(* IEC 61131-3 sources: OpenPLC-Simulator/openplc/OpenPLC/src (part 2) *)

(* ---- SIM_FB_RunTasks.st ---- *)
(* ============================================================
   SIM_FB_RunTasks.st — Simulate transporter task execution

   For each active transporter [1..3], checks whether a new task
   has been assigned (task_id <> running_task_id) and executes
   the full transport cycle:

     Phase 0  idle        — waiting for new task
     Phase 1  to_lift     — X-drive towards lift station
     Phase 2  lifting     — Z-lift sequence (stages 1-5)
     Phase 3  to_sink     — X-drive towards sink station
     Phase 4  sinking     — Z-sink sequence (stages 6-8)

   Also maintains current_station (nearest station) every cycle.

   Called once per PLC scan from PLC_PRG.
   ============================================================ *)

FUNCTION_BLOCK SIM_FB_RunTasks
VAR_INPUT
  i_run : BOOL;       (* enable — typically init_done *)
END_VAR
VAR_EXTERNAL CONSTANT
    TRANSPORTERS : INT;
END_VAR

VAR_EXTERNAL
  g_transporter  : ARRAY[1..TRANSPORTERS] OF STC_TRANSPORTER_T;
  g_stations     : ARRAY[101..125] OF STATION_T;
  g_cfg          : ARRAY[1..TRANSPORTERS] OF TRANSPORTER_CFG_T;
  g_move         : ARRAY[1..TRANSPORTERS] OF MOVE_TIMES_T;
END_VAR
VAR
  i            : INT;
  idx          : INT;
  (* Physics FB instances — one per transporter (MATIEC needs separate instances) *)
  fb_x1        : SIM_FB_XMotion;
  fb_x2        : SIM_FB_XMotion;
  fb_x3        : SIM_FB_XMotion;
  fb_z1        : SIM_FB_ZMotion;
  fb_z2        : SIM_FB_ZMotion;
  fb_z3        : SIM_FB_ZMotion;
  (* Station lookup *)
  lookup       : STC_FB_FindStation;
  (* Temp vars for VAR_IN_OUT passing *)
  tmp_x        : REAL;
  tmp_vx       : REAL;
  tmp_z        : REAL;
  tmp_zs       : INT;
  tmp_zt       : REAL;
  arrived_x    : BOOL;
  at_station   : BOOL;    (* TRUE only when actually at station, not just at drive limit *)
  arrived_z    : BOOL;
  station_type : INT;
  device_delay : REAL;
  drop_time    : REAL;
  (* Nearest-station calculation *)
  nearest_num  : INT;
  min_dist     : REAL;
  dx           : REAL;
  (* Time measurement instances *)
  tm1          : STC_FB_MeasureMoveTimes;
  tm2          : STC_FB_MeasureMoveTimes;
  tm3          : STC_FB_MeasureMoveTimes;
END_VAR

IF NOT i_run THEN
  RETURN;
END_IF;

FOR i := 1 TO TRANSPORTERS DO
  IF g_transporter[i].active THEN

  (* ── Phase 0 → 1: Accept new task ───────────────────────── *)
  IF (g_transporter[i].phase = 0)
     AND (g_transporter[i].task_id <> g_transporter[i].running_task_id) THEN
    g_transporter[i].running_task_id := g_transporter[i].task_id;
    lookup(station_number := g_transporter[i].lift_station);
    g_transporter[i].final_target_x := lookup.x_mm;
    g_transporter[i].phase := 1;
    g_transporter[i].z_stage := 0;
    g_transporter[i].z_timer_s := 0.0;

  (* ── Phase 1: Drive X towards lift station ──────────────── *)
  ELSIF g_transporter[i].phase = 1 THEN
    tmp_x  := g_transporter[i].x_mm;
    tmp_vx := g_transporter[i].vel_x;
    IF i = 1 THEN
      fb_x1(
        delta_t  := 0.02,
        x_target := g_transporter[i].final_target_x,
        x_min    := g_transporter[i].x_min_limit,
        x_max    := g_transporter[i].x_max_limit,
        v_max    := g_cfg[i].phys2d.x_max_mm_s,
        t_acc    := g_cfg[i].phys2d.x_accel_s,
        t_dec    := g_cfg[i].phys2d.x_decel_s,
        x_pos    := tmp_x,
        v_x      := tmp_vx
      );
      arrived_x := fb_x1.arrived;
    ELSIF i = 2 THEN
      fb_x2(
        delta_t  := 0.02,
        x_target := g_transporter[i].final_target_x,
        x_min    := g_transporter[i].x_min_limit,
        x_max    := g_transporter[i].x_max_limit,
        v_max    := g_cfg[i].phys2d.x_max_mm_s,
        t_acc    := g_cfg[i].phys2d.x_accel_s,
        t_dec    := g_cfg[i].phys2d.x_decel_s,
        x_pos    := tmp_x,
        v_x      := tmp_vx
      );
      arrived_x := fb_x2.arrived;
    ELSIF i = 3 THEN
      fb_x3(
        delta_t  := 0.02,
        x_target := g_transporter[i].final_target_x,
        x_min    := g_transporter[i].x_min_limit,
        x_max    := g_transporter[i].x_max_limit,
        v_max    := g_cfg[i].phys2d.x_max_mm_s,
        t_acc    := g_cfg[i].phys2d.x_accel_s,
        t_dec    := g_cfg[i].phys2d.x_decel_s,
        x_pos    := tmp_x,
        v_x      := tmp_vx
      );
      arrived_x := fb_x3.arrived;
    END_IF;
    g_transporter[i].x_mm  := tmp_x;
    g_transporter[i].vel_x := tmp_vx;

    (* Only transition when actually at station, not just at drive limit *)
    at_station := arrived_x
                  AND (ABS(g_transporter[i].x_mm - g_transporter[i].final_target_x) <= 6.0);
    IF at_station THEN
      g_transporter[i].current_station := g_transporter[i].lift_station;
      lookup(station_number := g_transporter[i].lift_station);
      device_delay := lookup.device_delay_s;
      drop_time    := lookup.dropping_time_s;
      g_transporter[i].z_timer_s := device_delay + drop_time;
      g_transporter[i].z_stage := 1;
      g_transporter[i].phase := 2;
    END_IF;
    (* If arrived_x but not at_station → at drive limit, wait for clearance *)

  (* ── Phase 2: Lift Z at lift station ────────────────────── *)
  ELSIF g_transporter[i].phase = 2 THEN
    lookup(station_number := g_transporter[i].lift_station);
    station_type := lookup.stype;
    tmp_z  := g_transporter[i].z_mm;
    tmp_zs := g_transporter[i].z_stage;
    tmp_zt := g_transporter[i].z_timer_s;
    IF i = 1 THEN
      fb_z1(
        delta_t       := 0.02,
        station_type  := station_type,
        z_total_mm    := g_cfg[i].phys2d.z_total_mm,
        z_slow_dry_mm := g_cfg[i].phys2d.z_slow_dry_mm,
        z_slow_wet_mm := g_cfg[i].phys2d.z_slow_wet_mm,
        z_slow_end_mm := g_cfg[i].phys2d.z_slow_end_mm,
        z_slow_mm_s   := g_cfg[i].phys2d.z_slow_mm_s,
        z_fast_mm_s   := g_cfg[i].phys2d.z_fast_mm_s,
        drip_delay_s  := g_cfg[i].phys2d.drip_delay_s,
        z_mm          := tmp_z,
        z_stage       := tmp_zs,
        z_timer_s     := tmp_zt
      );
      arrived_z := fb_z1.done;
    ELSIF i = 2 THEN
      fb_z2(
        delta_t       := 0.02,
        station_type  := station_type,
        z_total_mm    := g_cfg[i].phys2d.z_total_mm,
        z_slow_dry_mm := g_cfg[i].phys2d.z_slow_dry_mm,
        z_slow_wet_mm := g_cfg[i].phys2d.z_slow_wet_mm,
        z_slow_end_mm := g_cfg[i].phys2d.z_slow_end_mm,
        z_slow_mm_s   := g_cfg[i].phys2d.z_slow_mm_s,
        z_fast_mm_s   := g_cfg[i].phys2d.z_fast_mm_s,
        drip_delay_s  := g_cfg[i].phys2d.drip_delay_s,
        z_mm          := tmp_z,
        z_stage       := tmp_zs,
        z_timer_s     := tmp_zt
      );
      arrived_z := fb_z2.done;
    ELSIF i = 3 THEN
      fb_z3(
        delta_t       := 0.02,
        station_type  := station_type,
        z_total_mm    := g_cfg[i].phys2d.z_total_mm,
        z_slow_dry_mm := g_cfg[i].phys2d.z_slow_dry_mm,
        z_slow_wet_mm := g_cfg[i].phys2d.z_slow_wet_mm,
        z_slow_end_mm := g_cfg[i].phys2d.z_slow_end_mm,
        z_slow_mm_s   := g_cfg[i].phys2d.z_slow_mm_s,
        z_fast_mm_s   := g_cfg[i].phys2d.z_fast_mm_s,
        drip_delay_s  := g_cfg[i].phys2d.drip_delay_s,
        z_mm          := tmp_z,
        z_stage       := tmp_zs,
        z_timer_s     := tmp_zt
      );
      arrived_z := fb_z3.done;
    END_IF;
    g_transporter[i].z_mm      := tmp_z;
    g_transporter[i].z_stage   := tmp_zs;
    g_transporter[i].z_timer_s := tmp_zt;
    IF arrived_z THEN
      lookup(station_number := g_transporter[i].sink_station);
      g_transporter[i].final_target_x := lookup.x_mm;
      g_transporter[i].phase := 3;
    END_IF;

  (* ── Phase 3: Drive X towards sink station ─────────────── *)
  ELSIF g_transporter[i].phase = 3 THEN
    tmp_x  := g_transporter[i].x_mm;
    tmp_vx := g_transporter[i].vel_x;
    IF i = 1 THEN
      fb_x1(
        delta_t  := 0.02,
        x_target := g_transporter[i].final_target_x,
        x_min    := g_transporter[i].x_min_limit,
        x_max    := g_transporter[i].x_max_limit,
        v_max    := g_cfg[i].phys2d.x_max_mm_s,
        t_acc    := g_cfg[i].phys2d.x_accel_s,
        t_dec    := g_cfg[i].phys2d.x_decel_s,
        x_pos    := tmp_x,
        v_x      := tmp_vx
      );
      arrived_x := fb_x1.arrived;
    ELSIF i = 2 THEN
      fb_x2(
        delta_t  := 0.02,
        x_target := g_transporter[i].final_target_x,
        x_min    := g_transporter[i].x_min_limit,
        x_max    := g_transporter[i].x_max_limit,
        v_max    := g_cfg[i].phys2d.x_max_mm_s,
        t_acc    := g_cfg[i].phys2d.x_accel_s,
        t_dec    := g_cfg[i].phys2d.x_decel_s,
        x_pos    := tmp_x,
        v_x      := tmp_vx
      );
      arrived_x := fb_x2.arrived;
    ELSIF i = 3 THEN
      fb_x3(
        delta_t  := 0.02,
        x_target := g_transporter[i].final_target_x,
        x_min    := g_transporter[i].x_min_limit,
        x_max    := g_transporter[i].x_max_limit,
        v_max    := g_cfg[i].phys2d.x_max_mm_s,
        t_acc    := g_cfg[i].phys2d.x_accel_s,
        t_dec    := g_cfg[i].phys2d.x_decel_s,
        x_pos    := tmp_x,
        v_x      := tmp_vx
      );
      arrived_x := fb_x3.arrived;
    END_IF;
    g_transporter[i].x_mm  := tmp_x;
    g_transporter[i].vel_x := tmp_vx;

    (* Only transition when actually at station, not just at drive limit *)
    at_station := arrived_x
                  AND (ABS(g_transporter[i].x_mm - g_transporter[i].final_target_x) <= 6.0);
    IF at_station THEN
      g_transporter[i].current_station := g_transporter[i].sink_station;
      lookup(station_number := g_transporter[i].sink_station);
      device_delay := lookup.device_delay_s;
      g_transporter[i].z_timer_s := device_delay + g_cfg[i].phys2d.drip_delay_s;
      g_transporter[i].z_stage := 6;
      g_transporter[i].phase := 4;
    END_IF;
    (* If arrived_x but not at_station → at drive limit, wait for clearance *)

  (* ── Phase 4: Sink Z at sink station ───────────────────── *)
  ELSIF g_transporter[i].phase = 4 THEN
    lookup(station_number := g_transporter[i].sink_station);
    station_type := lookup.stype;
    tmp_z  := g_transporter[i].z_mm;
    tmp_zs := g_transporter[i].z_stage;
    tmp_zt := g_transporter[i].z_timer_s;
    IF i = 1 THEN
      fb_z1(
        delta_t       := 0.02,
        station_type  := station_type,
        z_total_mm    := g_cfg[i].phys2d.z_total_mm,
        z_slow_dry_mm := g_cfg[i].phys2d.z_slow_dry_mm,
        z_slow_wet_mm := g_cfg[i].phys2d.z_slow_wet_mm,
        z_slow_end_mm := g_cfg[i].phys2d.z_slow_end_mm,
        z_slow_mm_s   := g_cfg[i].phys2d.z_slow_mm_s,
        z_fast_mm_s   := g_cfg[i].phys2d.z_fast_mm_s,
        drip_delay_s  := g_cfg[i].phys2d.drip_delay_s,
        z_mm          := tmp_z,
        z_stage       := tmp_zs,
        z_timer_s     := tmp_zt
      );
      arrived_z := fb_z1.done;
    ELSIF i = 2 THEN
      fb_z2(
        delta_t       := 0.02,
        station_type  := station_type,
        z_total_mm    := g_cfg[i].phys2d.z_total_mm,
        z_slow_dry_mm := g_cfg[i].phys2d.z_slow_dry_mm,
        z_slow_wet_mm := g_cfg[i].phys2d.z_slow_wet_mm,
        z_slow_end_mm := g_cfg[i].phys2d.z_slow_end_mm,
        z_slow_mm_s   := g_cfg[i].phys2d.z_slow_mm_s,
        z_fast_mm_s   := g_cfg[i].phys2d.z_fast_mm_s,
        drip_delay_s  := g_cfg[i].phys2d.drip_delay_s,
        z_mm          := tmp_z,
        z_stage       := tmp_zs,
        z_timer_s     := tmp_zt
      );
      arrived_z := fb_z2.done;
    ELSIF i = 3 THEN
      fb_z3(
        delta_t       := 0.02,
        station_type  := station_type,
        z_total_mm    := g_cfg[i].phys2d.z_total_mm,
        z_slow_dry_mm := g_cfg[i].phys2d.z_slow_dry_mm,
        z_slow_wet_mm := g_cfg[i].phys2d.z_slow_wet_mm,
        z_slow_end_mm := g_cfg[i].phys2d.z_slow_end_mm,
        z_slow_mm_s   := g_cfg[i].phys2d.z_slow_mm_s,
        z_fast_mm_s   := g_cfg[i].phys2d.z_fast_mm_s,
        drip_delay_s  := g_cfg[i].phys2d.drip_delay_s,
        z_mm          := tmp_z,
        z_stage       := tmp_zs,
        z_timer_s     := tmp_zt
      );
      arrived_z := fb_z3.done;
    END_IF;
    g_transporter[i].z_mm      := tmp_z;
    g_transporter[i].z_stage   := tmp_zs;
    g_transporter[i].z_timer_s := tmp_zt;
    IF arrived_z THEN
      g_transporter[i].phase := 0;
    END_IF;
  END_IF;  (* ELSIF chain: phases 0→1→2→3→4 *)

  (* ── Phase 0 idle: drive back inside limits if outside ────── *)
  IF g_transporter[i].phase = 0 THEN
    tmp_x  := g_transporter[i].x_mm;
    tmp_vx := g_transporter[i].vel_x;
    (* Use current position as target — XMotion will clamp to nearest limit if outside *)
    IF i = 1 THEN
      fb_x1(
        delta_t  := 0.02,
        x_target := tmp_x,
        x_min    := g_transporter[i].x_min_limit,
        x_max    := g_transporter[i].x_max_limit,
        v_max    := g_cfg[i].phys2d.x_max_mm_s,
        t_acc    := g_cfg[i].phys2d.x_accel_s,
        t_dec    := g_cfg[i].phys2d.x_decel_s,
        x_pos    := tmp_x,
        v_x      := tmp_vx
      );
    ELSIF i = 2 THEN
      fb_x2(
        delta_t  := 0.02,
        x_target := tmp_x,
        x_min    := g_transporter[i].x_min_limit,
        x_max    := g_transporter[i].x_max_limit,
        v_max    := g_cfg[i].phys2d.x_max_mm_s,
        t_acc    := g_cfg[i].phys2d.x_accel_s,
        t_dec    := g_cfg[i].phys2d.x_decel_s,
        x_pos    := tmp_x,
        v_x      := tmp_vx
      );
    ELSIF i = 3 THEN
      fb_x3(
        delta_t  := 0.02,
        x_target := tmp_x,
        x_min    := g_transporter[i].x_min_limit,
        x_max    := g_transporter[i].x_max_limit,
        v_max    := g_cfg[i].phys2d.x_max_mm_s,
        t_acc    := g_cfg[i].phys2d.x_accel_s,
        t_dec    := g_cfg[i].phys2d.x_decel_s,
        x_pos    := tmp_x,
        v_x      := tmp_vx
      );
    END_IF;
    g_transporter[i].x_mm  := tmp_x;
    g_transporter[i].vel_x := tmp_vx;
  END_IF;

  (* ── Nearest station tracking ──────────────────────────── *)
  min_dist := 1.0e9;
  nearest_num := g_transporter[i].current_station;
  FOR idx := 101 TO 125 DO
    IF g_stations[idx].tank_id <> 0 THEN
      dx := g_stations[idx].x_position - g_transporter[i].x_mm;
      IF ABS(dx) < min_dist THEN
        min_dist := ABS(dx);
        nearest_num := idx;
      END_IF;
    END_IF;
  END_FOR;
  g_transporter[i].current_station := nearest_num;

  (* ── Measure move times (one instance per transporter) ──── *)
  IF i = 1 THEN
    tm1(t_id := 1, phase := g_transporter[1].phase, delta_t := 0.02,
        vel_x := g_transporter[1].vel_x, z_stage := g_transporter[1].z_stage,
        lift_stn := g_transporter[1].lift_station,
        sink_stn := g_transporter[1].sink_station,
        from_stn := g_transporter[1].current_station);
  ELSIF i = 2 THEN
    tm2(t_id := 2, phase := g_transporter[2].phase, delta_t := 0.02,
        vel_x := g_transporter[2].vel_x, z_stage := g_transporter[2].z_stage,
        lift_stn := g_transporter[2].lift_station,
        sink_stn := g_transporter[2].sink_station,
        from_stn := g_transporter[2].current_station);
  ELSIF i = 3 THEN
    tm3(t_id := 3, phase := g_transporter[3].phase, delta_t := 0.02,
        vel_x := g_transporter[3].vel_x, z_stage := g_transporter[3].z_stage,
        lift_stn := g_transporter[3].lift_station,
        sink_stn := g_transporter[3].sink_station,
        from_stn := g_transporter[3].current_station);
  END_IF;

  END_IF;  (* active *)
END_FOR;

END_FUNCTION_BLOCK

(* ---- SIM_FB_XMotion.st ---- *)
(* ============================================================
   SIM_FB_XMotion.st — Horizontal motion with accel / decel
   ============================================================ *)

FUNCTION_BLOCK SIM_FB_XMotion
VAR_INPUT
  delta_t  : REAL;
  x_target : REAL;
  x_min    : REAL;
  x_max    : REAL;
  v_max    : REAL;
  t_acc    : REAL;
  t_dec    : REAL;
END_VAR
VAR_IN_OUT
  x_pos : REAL;
  v_x   : REAL;
END_VAR
VAR_OUTPUT
  arrived : BOOL;
END_VAR
VAR
  drive_target : REAL;
  distance     : REAL;
  dir          : REAL;
  a_acc        : REAL;
  a_dec        : REAL;
  brake_dist   : REAL;
  new_vel      : REAL;
  travel       : REAL;
END_VAR
  IF (x_max > x_min) THEN
    IF x_pos < x_min THEN
      drive_target := x_min;
    ELSIF x_pos > x_max THEN
      drive_target := x_max;
    ELSE
      IF x_target < x_min THEN
        drive_target := x_min;
      ELSIF x_target > x_max THEN
        drive_target := x_max;
      ELSE
        drive_target := x_target;
      END_IF;
    END_IF;
  ELSE
    drive_target := x_target;
  END_IF;

  arrived := ABS(x_pos - drive_target) <= 3.0;
  IF arrived THEN
    x_pos := drive_target;
    v_x := 0.0;
    RETURN;
  END_IF;

  IF t_acc <= 0.0 THEN t_acc := 0.001; END_IF;
  IF t_dec <= 0.0 THEN t_dec := 0.001; END_IF;
  IF v_max < 0.0 THEN v_max := 0.0; END_IF;

  a_acc := v_max / t_acc;
  a_dec := v_max / t_dec;

  dir := 1.0;
  IF drive_target < x_pos THEN
    dir := -1.0;
  END_IF;

  distance := ABS(drive_target - x_pos);

  IF a_dec > 0.0 THEN
    brake_dist := (v_x * v_x) / (2.0 * a_dec);
  ELSE
    brake_dist := 0.0;
  END_IF;

  IF brake_dist >= distance THEN
    new_vel := v_x - a_dec * delta_t;
    IF new_vel < 0.0 THEN new_vel := 0.0; END_IF;
  ELSE
    new_vel := v_x + a_acc * delta_t;
    IF new_vel > v_max THEN new_vel := v_max; END_IF;
  END_IF;

  travel := new_vel * delta_t;
  IF travel >= distance THEN
    x_pos := drive_target;
    v_x := 0.0;
    arrived := TRUE;
  ELSE
    x_pos := x_pos + dir * travel;
    v_x := new_vel;
    arrived := FALSE;
  END_IF;
END_FUNCTION_BLOCK

(* ---- SIM_FB_ZMotion.st ---- *)
(* ============================================================
   SIM_FB_ZMotion.st — Vertical (Z) motion simulation

   Simulates 2D transporter lift/sink with realistic physics:
   - Slow start / fast middle / slow end speed profiles
   - Different slow zones for wet vs dry stations
   - Device delays and drip delays

   Coordinate convention: z=0 is bottom (sunk), z=z_total is top (lifted)

   LIFT sequence (z_stage 1-5):
     1: Init delay  (device_delay + dropping_time)
     2: Slow lift    0 → slow_zone
     3: Fast lift    → (z_total - z_slow_end_mm)
     4: Slow end     → z_total_mm
     5: Drip delay   at top position

   SINK sequence (z_stage 6-8):
     6: Init delay  (device_delay + drip_delay)
     7: Fast sink    z_total → slow_zone
     8: Slow sink    → 0 mm

   Caller sets z_stage and z_timer_s before first call.
   Output 'done' pulses TRUE when sequence completes.
   ============================================================ *)

FUNCTION_BLOCK SIM_FB_ZMotion
VAR_INPUT
  delta_t       : REAL;    (* Cycle time in seconds *)
  station_type  : INT;     (* STN_DRY=0, STN_WET=1 *)
  z_total_mm    : REAL;    (* Total Z travel distance *)
  z_slow_dry_mm : REAL;    (* Slow zone for dry stations *)
  z_slow_wet_mm : REAL;    (* Slow zone for wet stations *)
  z_slow_end_mm : REAL;    (* Slow zone at end of travel *)
  z_slow_mm_s   : REAL;    (* Slow speed mm/s *)
  z_fast_mm_s   : REAL;    (* Fast speed mm/s *)
  drip_delay_s  : REAL;    (* Drip delay after lift *)
END_VAR
VAR_IN_OUT
  z_mm      : REAL;        (* Current Z position *)
  z_stage   : INT;         (* Current motion stage *)
  z_timer_s : REAL;        (* Delay timer *)
END_VAR
VAR_OUTPUT
  done : BOOL;             (* TRUE when sequence complete *)
END_VAR
VAR_EXTERNAL CONSTANT
  STN_WET : INT;
END_VAR
VAR
  slow_zone : REAL;
END_VAR

  done := FALSE;

  (* Select slow zone based on station type *)
  IF station_type = STN_WET THEN
    slow_zone := z_slow_wet_mm;
  ELSE
    slow_zone := z_slow_dry_mm;
  END_IF;

  CASE z_stage OF

    (* === LIFT: stages 1-5 — nosto altaasta ylös (z kasvaa: 0 → z_total) === *)

    1: (* Init delay: device_delay + dropping_time *)
      z_timer_s := z_timer_s - delta_t;
      IF z_timer_s <= 0.0 THEN
        z_stage := 2;
        z_mm := 0.0;
      END_IF;

    2: (* Slow lift start — hidas nosto nesteestä *)
      z_mm := z_mm + z_slow_mm_s * delta_t;
      IF z_mm >= slow_zone THEN
        z_stage := 3;
      END_IF;

    3: (* Fast lift — nopea nosto *)
      z_mm := z_mm + z_fast_mm_s * delta_t;
      IF z_mm >= (z_total_mm - z_slow_end_mm) THEN
        z_stage := 4;
      END_IF;

    4: (* Slow lift end — hidas loppunosto *)
      z_mm := z_mm + z_slow_mm_s * delta_t;
      IF z_mm >= z_total_mm THEN
        z_mm := z_total_mm;
        z_timer_s := drip_delay_s;
        z_stage := 5;
      END_IF;

    5: (* Drip delay — tippumisviive yläasemassa *)
      z_timer_s := z_timer_s - delta_t;
      IF z_timer_s <= 0.0 THEN
        z_stage := 0;
        done := TRUE;
      END_IF;

    (* === SINK: stages 6-8 — lasku altaaseen (z pienenee: z_total → 0) === *)

    6: (* Init delay: device_delay + drip_delay *)
      z_timer_s := z_timer_s - delta_t;
      IF z_timer_s <= 0.0 THEN
        z_stage := 7;
      END_IF;

    7: (* Fast sink — nopea lasku *)
      z_mm := z_mm - z_fast_mm_s * delta_t;
      IF z_mm <= slow_zone THEN
        z_stage := 8;
      END_IF;

    8: (* Slow sink — hidas lasku nesteeseen *)
      z_mm := z_mm - z_slow_mm_s * delta_t;
      IF z_mm <= 0.0 THEN
        z_mm := 0.0;
        z_stage := 0;
        done := TRUE;
      END_IF;

  END_CASE;

END_FUNCTION_BLOCK

(* ---- STC_FB_CalcHorizontalTravel.st ---- *)
(* ============================================================
   STC_FB_CalcHorizontalTravel — Horizontal travel time (shared)
   ============================================================
   Calculates only the horizontal travel time between two stations
   (no lift/sink). Used for task sequence gap checks and departure
   idle-slot travel estimates.

   Logically stateless — implemented as FB because MATIEC does
   not allow VAR_EXTERNAL in FUNCTION.

   Used by: TSK_FB_Analyze (TASK_SEQUENCE check), DEP_*
   ============================================================ *)

FUNCTION_BLOCK STC_FB_CalcHorizontalTravel
VAR_INPUT
  i_from_stn : INT;     (* source station number *)
  i_to_stn   : INT;     (* destination station number *)
  i_trans    : INT;      (* transporter index 1..3 *)
END_VAR
VAR_OUTPUT
  o_travel_s : REAL;    (* horizontal travel time in seconds *)
END_VAR
VAR_EXTERNAL CONSTANT
    TRANSPORTERS : INT;
END_VAR

VAR_EXTERNAL
  g_move : ARRAY[1..TRANSPORTERS] OF MOVE_TIMES_T;
END_VAR
VAR
  from_idx : INT;
  to_idx   : INT;
END_VAR

o_travel_s := 0.0;
IF i_from_stn > 0 AND i_to_stn > 0 AND i_from_stn <> i_to_stn THEN
  from_idx := i_from_stn - 100;
  to_idx   := i_to_stn - 100;
  IF from_idx >= 1 AND from_idx <= 25 AND to_idx >= 1 AND to_idx <= 25
     AND i_trans >= 1 AND i_trans <= 3 THEN
    o_travel_s := g_move[i_trans].travel[from_idx].to_s[to_idx];
  END_IF;
END_IF;

END_FUNCTION_BLOCK

(* ---- STC_FB_CalcMoveTimes.st ---- *)
(* ============================================================
   STC_FB_CalcMoveTimes — Compute g_move from kinematic params
   ============================================================
   Calculates precomputed movement times for all active
   transporters using calibration kinematic parameters (g_cal)
   and station positions (g_station).

   For each transporter with valid g_cal data (x_max_mm_s > 0):
     - lift_s/sink_s: based on station kind (0=dry, 1=wet)
     - travel: trapezoidal velocity profile from X distances

   Call with i_run = TRUE to trigger computation (rising edge).

   Replaces need to re-run full calibration sequence when
   kinematic parameters are already known (e.g. loaded from
   a previously saved movement_times.json).
   ============================================================ *)

FUNCTION_BLOCK STC_FB_CalcMoveTimes
VAR_INPUT
  i_run : BOOL;    (* rising edge triggers computation *)
END_VAR
VAR_EXTERNAL CONSTANT
    MAX_Transporters    : INT;
    MIN_StationIndex : INT;
    MAX_StationIndex   : INT;
END_VAR
VAR_EXTERNAL
  g_cal           : ARRAY[1..MAX_Transporters] OF CALIBRATION_T;
  g_station       : ARRAY[MIN_StationIndex..MAX_StationIndex] OF UDT_StationType;
  g_move          : ARRAY[1..MAX_Transporters] OF MOVE_TIMES_T;
  g_station_count : INT;
END_VAR
VAR
  prev_run  : BOOL := FALSE;
  tid       : INT;
  si        : INT;
  sj        : INT;
  idx_i     : INT;
  idx_j     : INT;
  last_stn  : INT;    (* last active station number *)
  vm        : REAL;   (* max velocity mm/s *)
  ta        : REAL;   (* accel time s *)
  td        : REAL;   (* decel time s *)
  d_acc     : REAL;   (* accel distance mm *)
  d_dec     : REAL;   (* decel distance mm *)
  dist      : REAL;   (* distance between stations mm *)
  t_time    : REAL;   (* computed travel time *)
  v_peak    : REAL;   (* peak velocity in triangle profile *)
END_VAR

(* Rising edge detection *)
IF i_run AND NOT prev_run THEN

  (* Determine last active station *)
  last_stn := MIN_StationIndex + g_station_count - 1;
  IF last_stn > MAX_StationIndex THEN
    last_stn := MAX_StationIndex;
  END_IF;

  FOR tid := 1 TO MAX_Transporters DO
    (* Skip transporters without valid calibration data *)
    IF g_cal[tid].x_max_mm_s >= 1.0 THEN

      vm := g_cal[tid].x_max_mm_s;
      ta := g_cal[tid].x_accel_s;
      td := g_cal[tid].x_decel_s;
      d_acc := 0.5 * vm * ta;
      d_dec := 0.5 * vm * td;

      (* --- Lift and sink times per station --- *)
      FOR si := MIN_StationIndex TO last_stn DO
        idx_i := si - MIN_StationIndex + 1;
        IF idx_i >= 1 AND idx_i <= 30 THEN
          IF g_station[si].DryWet = 1 THEN
            (* Wet station *)
            g_move[tid].lift_s[idx_i] := g_cal[tid].lift_wet_s;
            g_move[tid].sink_s[idx_i] := g_cal[tid].sink_wet_s;
          ELSE
            (* Dry station *)
            g_move[tid].lift_s[idx_i] := g_cal[tid].lift_dry_s;
            g_move[tid].sink_s[idx_i] := g_cal[tid].sink_dry_s;
          END_IF;
        END_IF;
      END_FOR;

      (* --- Travel times between stations --- *)
      FOR si := MIN_StationIndex TO last_stn DO
        idx_i := si - MIN_StationIndex + 1;
        IF idx_i >= 1 AND idx_i <= 30 THEN
          FOR sj := MIN_StationIndex TO last_stn DO
            idx_j := sj - MIN_StationIndex + 1;
            IF idx_j >= 1 AND idx_j <= 30 THEN
              IF si = sj THEN
                g_move[tid].travel[idx_i].to_s[idx_j] := 0.0;
              ELSE
                dist := ABS(g_station[si].XPosition - g_station[sj].XPosition);
                IF dist < 1.0 THEN
                  t_time := 0.0;
                ELSIF dist >= d_acc + d_dec THEN
                  (* Trapezoidal profile: full accel + cruise + full decel *)
                  t_time := ta + (dist - d_acc - d_dec) / vm + td;
                ELSE
                  (* Triangle profile: cannot reach full speed *)
                  IF ta + td > 0.0 THEN
                    v_peak := SQRT(2.0 * dist * vm / (ta + td));
                    t_time := v_peak * (ta + td) / vm;
                  ELSE
                    t_time := 0.0;
                  END_IF;
                END_IF;
                g_move[tid].travel[idx_i].to_s[idx_j] := t_time;
              END_IF;
            END_IF;
          END_FOR;
        END_IF;
      END_FOR;

    END_IF;  (* valid calibration check *)
  END_FOR;

END_IF;

prev_run := i_run;

END_FUNCTION_BLOCK

(* ---- STC_FB_CalcTransferTime.st ---- *)
(* ============================================================
   STC_FB_CalcTransferTime — Transfer time calculation (shared)
   ============================================================
   Calculates total transfer time (lift + horizontal travel + sink)
   between two stations using precomputed g_move table.

   Logically stateless — implemented as FB because MATIEC does
   not allow VAR_EXTERNAL in FUNCTION.

   Used by: TSK_FB_CalcSchedule, TSK_FB_NoTreatment, DEP_*
   ============================================================ *)

FUNCTION_BLOCK STC_FB_CalcTransferTime
VAR_INPUT
  i_from_stn : INT;     (* source station, e.g. 105 *)
  i_to_stn   : INT;     (* destination station, e.g. 112 *)
  i_trans    : INT;      (* transporter index 1..3 *)
END_VAR
VAR_OUTPUT
  o_total_s  : REAL;    (* lift + travel + sink *)
  o_lift_s   : REAL;
  o_travel_s : REAL;
  o_sink_s   : REAL;
END_VAR
VAR_EXTERNAL CONSTANT
    TRANSPORTERS : INT;
END_VAR

VAR_EXTERNAL
  g_move : ARRAY[1..TRANSPORTERS] OF MOVE_TIMES_T;
END_VAR
VAR
  from_idx : INT;
  to_idx   : INT;
END_VAR

o_total_s  := 0.0;
o_lift_s   := 0.0;
o_travel_s := 0.0;
o_sink_s   := 0.0;

IF i_from_stn > 0 AND i_from_stn <> i_to_stn THEN
  from_idx := i_from_stn - 100;
  to_idx   := i_to_stn - 100;
  IF from_idx >= 1 AND from_idx <= 25 AND to_idx >= 1 AND to_idx <= 25
     AND i_trans >= 1 AND i_trans <= 3 THEN
    o_lift_s   := g_move[i_trans].lift_s[from_idx];
    o_travel_s := g_move[i_trans].travel[from_idx].to_s[to_idx];
    o_sink_s   := g_move[i_trans].sink_s[to_idx];
    o_total_s  := o_lift_s + o_travel_s + o_sink_s;
  END_IF;
END_IF;

END_FUNCTION_BLOCK

(* ---- STC_FB_Calibrate.st ---- *)
(* ============================================================
   STC_FB_Calibrate — Teaching / calibration mode
   ============================================================
   Runs 2 normal tasks per transporter to measure real lift,
   sink, and travel kinematic parameters.

   Task 1: lift=dry_station, sink=wet_station
     → MeasureMoveTimes records: lift_s[dry], sink_s[wet],
       travel[dry→wet]
     → X velocity profile measured during phase 3.

   Task 2: lift=wet_station, sink=dry_station
     → MeasureMoveTimes records: lift_s[wet], sink_s[dry],
       travel[wet→dry]

   Two tasks give ALL measurements: lift_wet, sink_wet,
   lift_dry, sink_dry, and X kinematics from vel profile.

   Calibration sequence per transporter:
     Step 10-12: Task 1 (dry→wet) + X velocity measurement
     Step 20-22: Task 2 (wet→dry)
     Step 30:    Read results from g_move → g_cal
     Step 40:    Next transporter or cal_step 100

   Global control:
     Step   0: Idle (waiting for cmd=1)
     Step 100: All measurement done (waiting for cmd=2 = Calculate)
     Step 200: Calculating g_move from measured parameters
     Step 999: Complete (waiting for cmd=3 = abort/reset)

   Inputs:
     i_run  — enable (typically init_done)
     i_cmd  — one-shot command: 1=start, 2=calculate, 3=abort

   Outputs:
     o_step   — current cal_step number
     o_tid    — transporter being calibrated
     o_active — TRUE while calibration is running
   ============================================================ *)

FUNCTION_BLOCK STC_FB_Calibrate
VAR_INPUT
  i_run : BOOL;       (* enable — typically init_done *)
  i_cmd : INT;        (* one-shot: 1=start, 2=calculate, 3=abort *)
END_VAR
VAR_OUTPUT
  o_step   : INT;     (* current calibration cal_step *)
  o_tid    : INT;     (* transporter being calibrated *)
  o_active : BOOL;    (* calibration in progress *)
END_VAR
VAR_EXTERNAL CONSTANT
    TRANSPORTERS : INT;
END_VAR

VAR_EXTERNAL
  g_transporter : ARRAY[1..TRANSPORTERS] OF STC_TRANSPORTER_T;
  g_stations    : ARRAY[101..125] OF STATION_T;
  g_cfg         : ARRAY[1..TRANSPORTERS] OF TRANSPORTER_CFG_T;
  g_cal         : ARRAY[1..TRANSPORTERS] OF CALIBRATION_T;
  g_move        : ARRAY[1..TRANSPORTERS] OF MOVE_TIMES_T;
  g_time_s      : LINT;
END_VAR
VAR
  cal_step       : INT := 0;
  tid        : INT := 0;      (* current transporter 1..3 *)
  task_key   : LINT := 0;   (* task_id for issued task *)
  (* X velocity measurement during phase 3 of task 1 *)
  x_meas_ph  : INT := 0;      (* 0=wait 1=accel 2=cruise 3=decel *)
  x_timer    : REAL := 0.0;
  x_prev_v   : REAL := 0.0;
  x_max_v    : REAL := 0.0;
  x_acc_t    : REAL := 0.0;
  x_dec_t    : REAL := 0.0;
  cur_v      : REAL;
  (* Calculation loop variables *)
  ci         : INT;
  cj         : INT;
  dist       : REAL;
  d_acc      : REAL;
  d_dec      : REAL;
  v_peak     : REAL;
  travel_t   : REAL;
  vm         : REAL;
  ta         : REAL;
  td         : REAL;
  (* Helper *)
  next_tid   : INT;
  wet_idx    : INT;
  dry_idx    : INT;
END_VAR

IF NOT i_run THEN
  RETURN;
END_IF;

(* ── Command handling ── *)
IF i_cmd = 1 AND cal_step = 0 THEN
  (* Start calibration — find first active transporter with plan *)
  tid := 0;
  FOR ci := 1 TO TRANSPORTERS DO
    IF g_transporter[ci].active AND tid = 0 THEN
      IF g_cal[ci].wet_station > 0 AND g_cal[ci].dry_station > 0 THEN
        tid := ci;
      END_IF;
    END_IF;
  END_FOR;
  IF tid > 0 THEN
    cal_step := 10;
    o_active := TRUE;
  END_IF;
END_IF;

IF i_cmd = 2 AND cal_step = 100 THEN
  (* Calculate g_move from measured parameters *)
  cal_step := 200;
END_IF;

IF i_cmd = 3 THEN
  (* Abort — reset to idle *)
  cal_step := 0;
  tid := 0;
  o_active := FALSE;
END_IF;

(* ================================================================
   STEP 10-12: TASK 1 — lift=dry_station, sink=wet_station
   MeasureMoveTimes records lift_s[dry], sink_s[wet], travel[dry→wet].
   X velocity profile measured during phase 3 (travel dry→wet).
   ================================================================ *)
IF cal_step = 10 THEN
  (* Issue task 1: lift from dry, sink to wet *)
  task_key := g_time_s;
  g_transporter[tid].task_id := task_key;
  g_transporter[tid].lift_station := g_cal[tid].dry_station;
  g_transporter[tid].sink_station := g_cal[tid].wet_station;
  (* Reset X velocity measurement *)
  x_meas_ph := 0;
  x_timer   := 0.0;
  x_prev_v  := 0.0;
  x_max_v   := 0.0;
  x_acc_t   := 0.0;
  x_dec_t   := 0.0;
  cal_step := 11;
END_IF;

IF cal_step = 11 THEN
  (* Wait for task acceptance *)
  IF g_transporter[tid].running_task_id = task_key THEN
    cal_step := 12;
  END_IF;
END_IF;

IF cal_step = 12 THEN
  cur_v := ABS(g_transporter[tid].vel_x);

  (* ── Track X velocity during phase 3 (travel dry→wet) ── *)
  IF g_transporter[tid].phase = 3 THEN
    IF x_meas_ph = 0 AND cur_v > 0.5 THEN
      (* Acceleration started *)
      x_meas_ph := 1;
      x_timer := 0.02;
      x_prev_v := cur_v;
      x_max_v := cur_v;

    ELSIF x_meas_ph = 1 THEN
      x_timer := x_timer + 0.02;
      IF cur_v > x_max_v THEN
        x_max_v := cur_v;
      END_IF;
      IF cur_v <= x_prev_v THEN
        (* Velocity stopped increasing → reached v_max *)
        x_acc_t := x_timer - 0.02;
        x_meas_ph := 2;
        x_timer := 0.0;
      END_IF;
      x_prev_v := cur_v;

    ELSIF x_meas_ph = 2 THEN
      (* Cruising — wait for deceleration *)
      IF cur_v < x_max_v - 1.0 THEN
        x_meas_ph := 3;
        x_timer := 0.02;
      END_IF;

    ELSIF x_meas_ph = 3 THEN
      x_timer := x_timer + 0.02;
    END_IF;
  END_IF;

  (* ── Phase 3 ended or phase 4 reached: store X results ── *)
  IF g_transporter[tid].phase >= 4 AND x_meas_ph >= 1 THEN
    IF x_meas_ph = 3 THEN
      x_dec_t := x_timer;
    END_IF;
    g_cal[tid].x_accel_s  := x_acc_t;
    g_cal[tid].x_decel_s  := x_dec_t;
    g_cal[tid].x_max_mm_s := x_max_v;
    (* Don't re-enter — set meas_ph to done *)
    x_meas_ph := 99;
  END_IF;

  (* ── Wait for full task completion (phase returns to 0) ── *)
  IF g_transporter[tid].phase = 0 AND x_meas_ph >= 99 THEN
    cal_step := 20;
  END_IF;
END_IF;

(* ================================================================
   STEP 20-22: TASK 2 — lift=wet_station, sink=dry_station
   MeasureMoveTimes records lift_s[wet], sink_s[dry], travel[wet→dry].
   ================================================================ *)
IF cal_step = 20 THEN
  (* Issue task 2: lift from wet, sink to dry *)
  task_key := g_time_s + LINT#1;
  g_transporter[tid].task_id := task_key;
  g_transporter[tid].lift_station := g_cal[tid].wet_station;
  g_transporter[tid].sink_station := g_cal[tid].dry_station;
  cal_step := 21;
END_IF;

IF cal_step = 21 THEN
  IF g_transporter[tid].running_task_id = task_key THEN
    cal_step := 22;
  END_IF;
END_IF;

IF cal_step = 22 THEN
  (* Wait for task completion *)
  IF g_transporter[tid].phase = 0 THEN
    cal_step := 30;
  END_IF;
END_IF;

(* ================================================================
   STEP 30: READ RESULTS FROM g_move → g_cal
   MeasureMoveTimes has recorded all 4 lift/sink times into g_move.
   ================================================================ *)
IF cal_step = 30 THEN
  wet_idx := g_cal[tid].wet_station - 100;
  dry_idx := g_cal[tid].dry_station - 100;

  IF wet_idx >= 1 AND wet_idx <= 25 THEN
    g_cal[tid].lift_wet_s := g_move[tid].lift_s[wet_idx];
    g_cal[tid].sink_wet_s := g_move[tid].sink_s[wet_idx];
  END_IF;

  IF dry_idx >= 1 AND dry_idx <= 25 THEN
    g_cal[tid].lift_dry_s := g_move[tid].lift_s[dry_idx];
    g_cal[tid].sink_dry_s := g_move[tid].sink_s[dry_idx];
  END_IF;

  cal_step := 40;
END_IF;

(* ================================================================
   STEP 40: TRANSPORTER DONE — advance to next or finish
   ================================================================ *)
IF cal_step = 40 THEN
  (* Find next active transporter after current tid with plan *)
  next_tid := 0;
  FOR ci := tid + 1 TO TRANSPORTERS DO
    IF g_transporter[ci].active AND next_tid = 0 THEN
      IF g_cal[ci].wet_station > 0 AND g_cal[ci].dry_station > 0 THEN
        next_tid := ci;
      END_IF;
    END_IF;
  END_FOR;

  IF next_tid > 0 THEN
    (* Calibrate next transporter *)
    tid := next_tid;
    cal_step := 10;
  ELSE
    (* All transporters done — measurement complete *)
    cal_step := 100;
  END_IF;
END_IF;

(* ================================================================
   STEP 200: CALCULATE g_move FROM MEASURED PARAMETERS
   For each active transporter with calibration data:
     - Copy lift/sink wet times to all wet stations
     - Copy lift/sink dry times to all dry stations
     - Calculate all station-to-station travel times using
       measured v_max, t_acc, t_dec and station distances
   ================================================================ *)
IF cal_step = 200 THEN
  FOR ci := 1 TO TRANSPORTERS DO
    IF g_transporter[ci].active AND g_cal[ci].x_max_mm_s > 0.0 THEN

      vm := g_cal[ci].x_max_mm_s;
      ta := g_cal[ci].x_accel_s;
      td := g_cal[ci].x_decel_s;

      (* --- Fill lift_s and sink_s per station type --- *)
      FOR cj := 1 TO 25 DO
        IF g_stations[100 + cj].tank_id <> 0 THEN
          IF g_stations[100 + cj].stn_type = 1 THEN
            (* Wet station *)
            g_move[ci].lift_s[cj] := g_cal[ci].lift_wet_s;
            g_move[ci].sink_s[cj] := g_cal[ci].sink_wet_s;
          ELSE
            (* Dry station *)
            g_move[ci].lift_s[cj] := g_cal[ci].lift_dry_s;
            g_move[ci].sink_s[cj] := g_cal[ci].sink_dry_s;
          END_IF;
        END_IF;
      END_FOR;

      (* --- Calculate all travel times from kinematics --- *)
      (* d_acc = 0.5 * v_max * t_acc (distance during acceleration)
         d_dec = 0.5 * v_max * t_dec (distance during deceleration)
         If dist >= d_acc + d_dec:
           travel = t_acc + (dist - d_acc - d_dec) / v_max + t_dec
         Else (triangle profile):
           v_peak = SQRT(2 * dist * v_max / (t_acc + t_dec))
           travel = v_peak * (t_acc + t_dec) / v_max *)
      d_acc := 0.5 * vm * ta;
      d_dec := 0.5 * vm * td;

      FOR cj := 1 TO 25 DO
        IF g_stations[100 + cj].tank_id <> 0 THEN
          FOR wet_idx := 1 TO 25 DO
            IF g_stations[100 + wet_idx].tank_id <> 0 THEN
              IF cj = wet_idx THEN
                g_move[ci].travel[cj].to_s[wet_idx] := 0.0;
              ELSE
                dist := ABS(g_stations[100 + cj].x_position - g_stations[100 + wet_idx].x_position);
                IF dist < 1.0 THEN
                  g_move[ci].travel[cj].to_s[wet_idx] := 0.0;
                ELSIF dist >= (d_acc + d_dec) THEN
                  (* Full trapezoidal profile *)
                  travel_t := ta + (dist - d_acc - d_dec) / vm + td;
                  g_move[ci].travel[cj].to_s[wet_idx] := travel_t;
                ELSE
                  (* Triangle profile — cannot reach full speed *)
                  IF (ta + td) > 0.0 THEN
                    v_peak := SQRT(2.0 * dist * vm / (ta + td));
                    travel_t := v_peak * (ta + td) / vm;
                    g_move[ci].travel[cj].to_s[wet_idx] := travel_t;
                  ELSE
                    g_move[ci].travel[cj].to_s[wet_idx] := 0.0;
                  END_IF;
                END_IF;
              END_IF;
            END_IF;
          END_FOR;
        END_IF;
      END_FOR;

    END_IF;
  END_FOR;

  cal_step := 999;
END_IF;

(* ── Update outputs ── *)
o_step := cal_step;
o_tid  := tid;
IF cal_step > 0 AND cal_step < 999 THEN
  o_active := TRUE;
ELSIF cal_step = 999 THEN
  o_active := FALSE;
ELSE
  o_active := FALSE;
END_IF;

END_FUNCTION_BLOCK

(* ---- STC_FB_ClearTaskQueues.st ---- *)
(* ============================================================
   STC_FB_ClearTaskQueues — Zero-out all transporter task queues
   ============================================================
   Clears count and all 9 fields of each slot in g_tasks[1..3].

   Replaces 2× identical clear loops in:
     TSK_FB_Scheduler (phase 2000)
     DEP_FB_Scheduler (phase 1020)
   ============================================================ *)

FUNCTION_BLOCK STC_FB_ClearTaskQueues
VAR_EXTERNAL CONSTANT
    TRANSPORTERS : INT;
END_VAR

VAR_EXTERNAL
  g_tasks : ARRAY[1..TRANSPORTERS] OF TSK_QUEUE_T;
END_VAR
VAR
  ti : INT;
  qi : INT;
END_VAR

FOR ti := 1 TO TRANSPORTERS DO
  g_tasks[ti].count := 0;
  FOR qi := 1 TO 10 DO
    g_tasks[ti].queue[qi].unit         := 0;
    g_tasks[ti].queue[qi].stage        := 0;
    g_tasks[ti].queue[qi].lift_station := 0;
    g_tasks[ti].queue[qi].sink_station := 0;
    g_tasks[ti].queue[qi].start_time   := 0;
    g_tasks[ti].queue[qi].finish_time  := 0;
    g_tasks[ti].queue[qi].calc_time    := 0.0;
    g_tasks[ti].queue[qi].min_time     := 0.0;
    g_tasks[ti].queue[qi].max_time     := 0.0;
  END_FOR;
END_FOR;

END_FUNCTION_BLOCK

(* ---- STC_FB_CollectActiveBatches.st ---- *)
(* ============================================================
   STC_FB_CollectActiveBatches — Filter active batches to list
   ============================================================
   Scans g_batch[1..10] and collects unit indices matching
   mode-specific conditions into an output list.

   Common conditions for both modes:
     unit.Status  = USED (1)
     unit.target  = TO_NONE (0)
     batch.prog_id = g_program[ui].program_id  (valid program)

   Mode:
     i_mode = 0 — active (in-production) batches:
                   batch.state = IN_PROCESS (1)
                   batch.cur_stage >= 0 AND <= 99
     i_mode = 1 — waiting batches:
                   batch.state = NOT_PROCESSED (0)

   Replaces 3× duplicated collection loops in:
     TSK_FB_Scheduler (phase 1, active batches)
     DEP_FB_Scheduler (phase 100, active + waiting batches)
   ============================================================ *)

FUNCTION_BLOCK STC_FB_CollectActiveBatches
VAR_INPUT
  i_mode : INT;    (* 0 = all active, 1 = waiting only *)
END_VAR
VAR_EXTERNAL CONSTANT
    MAX_Units : INT;
END_VAR
VAR_EXTERNAL
  g_batch   : ARRAY[1..MAX_Units] OF UDT_BatchType;
  g_unit    : ARRAY[1..MAX_Units] OF UDT_UnitType;
  g_program : ARRAY[1..MAX_Units] OF UDT_TreatmentProgramType;
END_VAR
VAR_OUTPUT
  o_list  : ARRAY[1..MAX_Units] OF INT;  (* unit indices *)
  o_count : INT;
END_VAR
VAR
  ui : INT;
END_VAR

o_count := 0;
FOR ui := 1 TO MAX_Units DO
  o_list[ui] := 0;
END_FOR;

FOR ui := 1 TO MAX_Units DO
  (* Common conditions: unit USED, target TO_NONE, valid program *)
  IF g_unit[ui].Status = 1
     AND g_unit[ui].target = 0
     AND g_batch[ui].prog_id = g_program[ui].program_id
     AND g_program[ui].program_id > 0 THEN

    IF i_mode = 0 THEN
      (* Active batches: IN_PROCESS, stage 0..99 *)
      IF g_batch[ui].state = 1
         AND g_batch[ui].cur_stage >= 0
         AND g_batch[ui].cur_stage <= 99 THEN
        o_count := o_count + 1;
        o_list[o_count] := ui;
      END_IF;
    ELSIF i_mode = 1 THEN
      (* Waiting batches: NOT_PROCESSED *)
      IF g_batch[ui].state = 0 THEN
        o_count := o_count + 1;
        o_list[o_count] := ui;
      END_IF;
    END_IF;
  END_IF;
END_FOR;

END_FUNCTION_BLOCK

(* ---- STC_FB_DispatchTask.st ---- *)
(* ============================================================
   STC_FB_DispatchTask — Validate and dispatch tasks to transporters
   ============================================================
   Called every PLC scan from MainScheduler (before TSK/DEP).
   For each idle transporter with queued tasks:

     1. Skip if transporter not idle (phase <> 0) or queue empty
     2. Time check: is start_time close enough?
        travel_time_to_lift + 3s >= time_until_start → proceed
     3. Sink station free check:
        a) Original sink free → use it
        b) Not free → search alternative parallel stations
           (from g_program[].stages[] or g_ntt[] for stage=0)
        c) Pick the station with oldest change_time (longest empty)
        d) No free alternative → skip, don't dispatch
     4. Conflict check: no other active transporter targeting
        same lift or sink station
     5. Dispatch: write task_id, lift_station, sink_station
        to g_transporter → RunTasks picks it up

   Used by: STC_FB_MainScheduler
   ============================================================ *)

FUNCTION_BLOCK STC_FB_DispatchTask
VAR_EXTERNAL CONSTANT
    MAX_TRANSPORTERS    : INT;
    MAX_UNITS           : INT;
    MAX_PARALLELS       : INT;
    MAX_STAGES          : INT;
    STATION_ARRAY_START : INT;
    STATION_ARRAY_END   : INT;
END_VAR
VAR_EXTERNAL
  g_transporter : ARRAY[1..MAX_TRANSPORTERS] OF STC_TRANSPORTER_T;
  g_task        : ARRAY[1..MAX_TRANSPORTERS] OF TSK_QUEUE_T;
  g_station     : ARRAY[STATION_ARRAY_START..STATION_ARRAY_END] OF STATION_T;
  g_unit        : ARRAY[1..MAX_UNITS] OF UNIT_T;
  g_program     : ARRAY[1..MAX_UNITS] OF TREATMENT_PROGRAM_T;
  g_ntt         : ARRAY[1..MAX_TRANSPORTERS] OF NTT_TRANSPORTER_T;
  g_batch       : ARRAY[1..MAX_UNITS] OF BATCH_T;
  g_move        : ARRAY[1..MAX_TRANSPORTERS] OF MOVE_TIMES_T;
  g_time_s      : LINT;
END_VAR
VAR
  ti           : INT;     (* transporter loop *)
  (* Task fields — read from queue[1] to avoid struct copy *)
  t_unit       : INT;
  t_stage      : INT;
  t_lift       : INT;
  t_sink       : INT;
  t_start      : LINT;
  t_calc_time  : REAL;
  (* Time check *)
  travel_s     : REAL;
  margin_s     : LINT;
  from_idx     : INT;
  to_idx       : INT;
  (* Sink search *)
  sink_stn     : INT;
  sink_free    : BOOL;
  best_stn     : INT;
  best_change  : LINT;
  si           : INT;
  cand_stn     : INT;
  cand_free    : BOOL;
  uj           : INT;
  tgt          : INT;
  ntt_idx      : INT;     (* resolved NTT index (buffer 6/7/8) *)
  ntt_cnt      : INT;
  ntt_fb_cnt   : INT;
  (* Conflict check *)
  conflict     : BOOL;
  cj           : INT;
  task_min     : INT;     (* min station of our proposed task *)
  task_max     : INT;     (* max station of our proposed task *)
  (* Shift-down after dispatch *)
  sh           : INT;
END_VAR

FOR ti := 1 TO MAX_TRANSPORTERS DO

  (* ── 1. Skip if not idle or queue empty ── *)
  IF g_transporter[ti].phase = 0 AND g_task[ti].count >= 1 THEN

    (* Read task fields from queue position 1 *)
    t_unit      := g_task[ti].queue[1].unit;
    t_stage     := g_task[ti].queue[1].stage;
    t_lift      := g_task[ti].queue[1].lift_station;
    t_sink      := g_task[ti].queue[1].sink_station;
    t_start     := g_task[ti].queue[1].start_time;
    t_calc_time := g_task[ti].queue[1].calc_time;

    (* ── 2. Time check ── *)
    travel_s := 0.0;
    IF g_transporter[ti].current_station > 0 AND t_lift > 0
       AND g_transporter[ti].current_station <> t_lift THEN
      from_idx := g_transporter[ti].current_station - 100;
      to_idx   := t_lift - 100;
      IF from_idx >= 1 AND from_idx <= 30 AND to_idx >= 1 AND to_idx <= 30 THEN
        travel_s := g_move[ti].travel[from_idx].to_s[to_idx];
      END_IF;
    END_IF;

    margin_s := t_start - g_time_s;

    IF margin_s <= REAL_TO_LINT(travel_s) + 3 THEN

      (* ── 3. Sink station free check ── *)
      sink_stn := t_sink;
      sink_free := FALSE;

      IF sink_stn >= STATION_ARRAY_START AND sink_stn <= STATION_ARRAY_END THEN
        sink_free := TRUE;
        FOR uj := 1 TO MAX_UNITS DO
          IF g_unit[uj].location = sink_stn AND g_unit[uj].status = 1 THEN
            sink_free := FALSE;
          END_IF;
        END_FOR;
      END_IF;

      IF NOT sink_free THEN
        (* Search alternative parallel stations *)
        best_stn := 0;
        best_change := LINT#2000000000;

        IF t_stage >= 1 AND t_stage <= MAX_STAGES
           AND t_unit >= 1 AND t_unit <= MAX_UNITS THEN
          (* Treatment task — look in g_program for parallel stations *)
          FOR si := 1 TO MAX_PARALLELS DO
            cand_stn := g_program[t_unit].stages[t_stage].stations[si];
            IF cand_stn > 0 AND cand_stn <> t_sink THEN
              IF cand_stn >= STATION_ARRAY_START AND cand_stn <= STATION_ARRAY_END THEN
                cand_free := TRUE;
                FOR uj := 1 TO MAX_UNITS DO
                  IF g_unit[uj].location = cand_stn AND g_unit[uj].status = 1 THEN
                    cand_free := FALSE;
                  END_IF;
                END_FOR;
                IF cand_free THEN
                  IF g_station[cand_stn].change_time < best_change THEN
                    best_change := g_station[cand_stn].change_time;
                    best_stn := cand_stn;
                  END_IF;
                END_IF;
              END_IF;
            END_IF;
          END_FOR;

        ELSIF t_stage = 0 AND t_unit >= 1 AND t_unit <= MAX_UNITS THEN
          (* No-treatment task — look in g_ntt for alternatives *)
          tgt := g_unit[t_unit].target;
          IF tgt >= 1 AND tgt <= 5 THEN
            (* Resolve buffer NTT index like NoTreatment does *)
            IF tgt = 2 THEN
              IF g_batch[t_unit].batch_code = 0 THEN
                ntt_idx := 6;
              ELSIF g_batch[t_unit].state = 2 THEN
                ntt_idx := 8;
              ELSE
                ntt_idx := 7;
              END_IF;
            ELSE
              ntt_idx := tgt;
            END_IF;
            (* Check primary stations *)
            ntt_cnt := g_ntt[ti].target[ntt_idx].station_count;
            FOR si := 1 TO ntt_cnt DO
              IF si <= MAX_PARALLELS THEN
                cand_stn := g_ntt[ti].target[ntt_idx].stations[si];
                IF cand_stn > 0 AND cand_stn <> t_sink THEN
                  IF cand_stn >= STATION_ARRAY_START AND cand_stn <= STATION_ARRAY_END THEN
                    cand_free := TRUE;
                    FOR uj := 1 TO MAX_UNITS DO
                      IF g_unit[uj].location = cand_stn AND g_unit[uj].status = 1 THEN
                        cand_free := FALSE;
                      END_IF;
                    END_FOR;
                    IF cand_free THEN
                      IF g_station[cand_stn].change_time < best_change THEN
                        best_change := g_station[cand_stn].change_time;
                        best_stn := cand_stn;
                      END_IF;
                    END_IF;
                  END_IF;
                END_IF;
              END_IF;
            END_FOR;
            (* Check fallback stations *)
            ntt_fb_cnt := g_ntt[ti].target[ntt_idx].fallback_count;
            FOR si := 1 TO ntt_fb_cnt DO
              IF si <= MAX_PARALLELS THEN
                cand_stn := g_ntt[ti].target[ntt_idx].fallback_stations[si];
                IF cand_stn > 0 AND cand_stn <> t_sink THEN
                  IF cand_stn >= STATION_ARRAY_START AND cand_stn <= STATION_ARRAY_END THEN
                    cand_free := TRUE;
                    FOR uj := 1 TO MAX_UNITS DO
                      IF g_unit[uj].location = cand_stn AND g_unit[uj].status = 1 THEN
                        cand_free := FALSE;
                      END_IF;
                    END_FOR;
                    IF cand_free THEN
                      IF g_station[cand_stn].change_time < best_change THEN
                        best_change := g_station[cand_stn].change_time;
                        best_stn := cand_stn;
                      END_IF;
                    END_IF;
                  END_IF;
                END_IF;
              END_IF;
            END_FOR;
          END_IF;
        END_IF;

        IF best_stn > 0 THEN
          sink_stn := best_stn;
          sink_free := TRUE;
        END_IF;
      END_IF;  (* NOT sink_free *)

      IF sink_free THEN

        (* ── 4. Conflict check ── *)
        (* Check against other transporters' ACTIVE tasks (phase>0).
           Two rules:
           a) T2's entire task (lift AND sink) is inside our task
              range [task_min..task_max] → conflict.
              Example: our 114→101 range [101,114]
                T2 114→113: both in [101,114] → conflict
                T2 114→117: 117 outside     → no conflict (going away)
           b) T2 delivers (sink) to one of our exact stations
              from outside our range → conflict.
              Example: T2 120→114, 114 is our lift → conflict *)
        conflict := FALSE;

        IF t_lift <= sink_stn THEN
          task_min := t_lift;
          task_max := sink_stn;
        ELSE
          task_min := sink_stn;
          task_max := t_lift;
        END_IF;

        FOR cj := 1 TO MAX_TRANSPORTERS DO
          IF cj <> ti AND g_transporter[cj].phase > 0 THEN

            (* a) T2's entire active task inside our range → conflict *)
            IF g_transporter[cj].lift_station >= task_min
               AND g_transporter[cj].lift_station <= task_max
               AND g_transporter[cj].sink_station >= task_min
               AND g_transporter[cj].sink_station <= task_max THEN
              conflict := TRUE;
            END_IF;

            (* b) T2 delivers to one of our exact stations → conflict *)
            IF g_transporter[cj].sink_station = t_lift
               OR g_transporter[cj].sink_station = sink_stn THEN
              conflict := TRUE;
            END_IF;

          END_IF;
        END_FOR;

        IF NOT conflict THEN
          (* ── 5. Dispatch: assign task to transporter ── *)
          g_transporter[ti].task_id      := t_start;
          g_transporter[ti].lift_station := t_lift;
          g_transporter[ti].sink_station := sink_stn;
          g_transporter[ti].unit_id      := t_unit;
          g_transporter[ti].treatment_time := t_calc_time;
          g_transporter[ti].remaining_time := t_calc_time;

          (* Copy station-specific timing from config *)
          IF t_lift >= STATION_ARRAY_START AND t_lift <= STATION_ARRAY_END THEN
            g_transporter[ti].dropping_time := g_station[t_lift].dropping_time;
            g_transporter[ti].lift_device_delay := g_station[t_lift].device_delay;
          END_IF;
          IF sink_stn >= STATION_ARRAY_START AND sink_stn <= STATION_ARRAY_END THEN
            g_transporter[ti].sink_device_delay := g_station[sink_stn].device_delay;
          END_IF;

          (* Shift queue: remove position 1, move rest up *)
          FOR sh := 2 TO g_task[ti].count DO
            g_task[ti].queue[sh - 1] := g_task[ti].queue[sh];
          END_FOR;
          (* Clear last slot *)
          g_task[ti].queue[g_task[ti].count].unit := 0;
          g_task[ti].queue[g_task[ti].count].stage := 0;
          g_task[ti].queue[g_task[ti].count].lift_station := 0;
          g_task[ti].queue[g_task[ti].count].sink_station := 0;
          g_task[ti].queue[g_task[ti].count].start_time := 0;
          g_task[ti].queue[g_task[ti].count].finish_time := 0;
          g_task[ti].queue[g_task[ti].count].calc_time := 0.0;
          g_task[ti].queue[g_task[ti].count].min_time := 0.0;
          g_task[ti].queue[g_task[ti].count].max_time := 0.0;
          g_task[ti].count := g_task[ti].count - 1;

        END_IF;  (* NOT conflict *)

      END_IF;  (* sink_free *)

    END_IF;  (* time check *)

  END_IF;  (* idle + queue *)

END_FOR;

END_FUNCTION_BLOCK

(* ---- STC_FB_EventQueue.st ---- *)
(* ============================================================
   STC_FB_EventQueue — Generic event message queue handler
   ============================================================
   Manages a circular 10-slot event queue (g_event) and the
   Modbus handshake with Gateway.

   - enqueue: caller writes msg fields to g_event_pending,
     then sets g_event_pending_valid := TRUE.
     This FB picks it up and adds to queue.
   - dequeue: copies head message to QW Modbus registers.
     Gateway reads, writes ack_seq back via IW.
     On ack match → advance head, count--.

   Called every PLC scan from plc_prg (always, not gated by
   scheduler turn).

   Handshake protocol:
     PLC:  qw_event_out_count, qw_event_out_seq, qw_event_out_type,
           qw_event_out_ts_hi/lo, qw_event_out_f1..f12 → Modbus holding regs
     GW:   iw_event_ack_seq → Modbus input register
     When qw_event_out_seq = iw_event_ack_seq: message consumed → next.
   ============================================================ *)

FUNCTION_BLOCK STC_FB_EventQueue
VAR_EXTERNAL
  g_event          : EVENT_QUEUE_T;
  (* Pending message — set by other FBs, consumed here *)
  g_event_pending       : EVENT_MSG_T;
  g_event_pending_valid : BOOL;
  (* Modbus output — head message visible to gateway *)
  qw_event_out_count   : INT;
  qw_event_out_seq     : INT;
  qw_event_out_type    : INT;
  qw_event_out_ts_hi   : INT;
  qw_event_out_ts_lo   : INT;
  qw_event_out_f1      : INT;
  qw_event_out_f2      : INT;
  qw_event_out_f3      : INT;
  qw_event_out_f4      : INT;
  qw_event_out_f5      : INT;
  qw_event_out_f6      : INT;
  qw_event_out_f7      : INT;
  qw_event_out_f8      : INT;
  qw_event_out_f9      : INT;
  qw_event_out_f10     : INT;
  qw_event_out_f11     : INT;
  qw_event_out_f12     : INT;
  (* Modbus input — gateway ack *)
  iw_event_ack_seq     : INT;
END_VAR
VAR
  tail : INT;   (* insertion index *)
END_VAR

(* ── 1. Enqueue: pick up pending message if queue not full ── *)
IF g_event_pending_valid AND g_event.count < 10 THEN
  (* Calculate tail position in circular buffer *)
  tail := ((g_event.head - 1 + g_event.count) MOD 10) + 1;

  (* Assign sequence number *)
  g_event_pending.seq := g_event.next_seq;
  g_event.next_seq := g_event.next_seq + 1;
  IF g_event.next_seq > 32000 THEN
    g_event.next_seq := 1;  (* wrap to avoid INT overflow *)
  END_IF;

  (* Store in buffer *)
  g_event.buf[tail] := g_event_pending;
  g_event.count := g_event.count + 1;

  (* Clear pending flag *)
  g_event_pending_valid := FALSE;
END_IF;

(* ── 2. Dequeue: check gateway ack for head message ── *)
IF g_event.count > 0 THEN
  IF iw_event_ack_seq = g_event.buf[g_event.head].seq THEN
    (* Gateway consumed this message — advance head *)
    g_event.head := (g_event.head MOD 10) + 1;
    g_event.count := g_event.count - 1;
  END_IF;
END_IF;

(* ── 3. Publish: copy head message to Modbus QW registers ── *)
qw_event_out_count := g_event.count;

IF g_event.count > 0 THEN
  qw_event_out_seq    := g_event.buf[g_event.head].seq;
  qw_event_out_type   := g_event.buf[g_event.head].msg_type;
  qw_event_out_ts_hi  := g_event.buf[g_event.head].ts_hi;
  qw_event_out_ts_lo  := g_event.buf[g_event.head].ts_lo;
  qw_event_out_f1     := g_event.buf[g_event.head].f[1];
  qw_event_out_f2     := g_event.buf[g_event.head].f[2];
  qw_event_out_f3     := g_event.buf[g_event.head].f[3];
  qw_event_out_f4     := g_event.buf[g_event.head].f[4];
  qw_event_out_f5     := g_event.buf[g_event.head].f[5];
  qw_event_out_f6     := g_event.buf[g_event.head].f[6];
  qw_event_out_f7     := g_event.buf[g_event.head].f[7];
  qw_event_out_f8     := g_event.buf[g_event.head].f[8];
  qw_event_out_f9     := g_event.buf[g_event.head].f[9];
  qw_event_out_f10    := g_event.buf[g_event.head].f[10];
  qw_event_out_f11    := g_event.buf[g_event.head].f[11];
  qw_event_out_f12    := g_event.buf[g_event.head].f[12];
ELSE
  (* Queue empty — clear output *)
  qw_event_out_seq    := 0;
  qw_event_out_type   := 0;
  qw_event_out_ts_hi  := 0;
  qw_event_out_ts_lo  := 0;
  qw_event_out_f1     := 0;
  qw_event_out_f2     := 0;
  qw_event_out_f3     := 0;
  qw_event_out_f4     := 0;
  qw_event_out_f5     := 0;
  qw_event_out_f6     := 0;
  qw_event_out_f7     := 0;
  qw_event_out_f8     := 0;
  qw_event_out_f9     := 0;
  qw_event_out_f10    := 0;
  qw_event_out_f11    := 0;
  qw_event_out_f12    := 0;
END_IF;

END_FUNCTION_BLOCK

(* ---- STC_FB_FindStation.st ---- *)
(* ============================================================
   fb_station_lookup.st → STC_FB_FindStation — Find a station by its number
   ============================================================ *)

FUNCTION_BLOCK STC_FB_FindStation
VAR_INPUT
  station_number : INT;
END_VAR
VAR_OUTPUT
  found           : BOOL;
  idx             : INT;
  x_mm            : REAL;
  stype           : INT;
  device_delay_s  : REAL;
  dropping_time_s : REAL;
END_VAR
VAR_EXTERNAL
  g_station : ARRAY[101..125] OF STATION_T;
END_VAR
VAR
  st : STATION_T;
END_VAR
  (* Direct lookup by station number — no loop needed *)
  IF (station_number >= 101) AND (station_number <= 125) THEN
    st := g_station[station_number];
    IF st.tank_id <> 0 THEN
      found := TRUE;
      idx := station_number;
      x_mm := st.x_position;
      stype := st.stn_type;
      device_delay_s := st.device_delay;
      dropping_time_s := st.dropping_time;
      RETURN;
    END_IF;
  END_IF;

  found := FALSE;
  idx := 0;
  x_mm := 0.0;
  stype := 0;
  device_delay_s := 0.0;
  dropping_time_s := 0.0;
END_FUNCTION_BLOCK

(* ---- STC_FB_FindTransporter.st ---- *)
(* ============================================================
   STC_FB_FindTransporter — Find covering transporter (shared)
   ============================================================
   Finds which transporter (1..3) can handle a lift→sink pair
   by checking g_cfg[].task_area[] coverage.

   If i_sink_stn = 0, only lift coverage is checked (used when
   looking for the transporter covering a single station).

   Logically stateless — implemented as FB because MATIEC does
   not allow VAR_EXTERNAL in FUNCTION.

   Used by: TSK_FB_CreateTasks, TSK_FB_NoTreatment,
            TSK_FB_Scheduler, DEP_*
   ============================================================ *)

FUNCTION_BLOCK STC_FB_FindTransporter
VAR_INPUT
  i_lift_stn : INT;     (* lift station number *)
  i_sink_stn : INT;     (* sink station number, 0 = lift-only search *)
END_VAR
VAR_OUTPUT
  o_trans_id : INT;     (* found transporter 1..3, 0 = not found *)
END_VAR
VAR_EXTERNAL CONSTANT
    TRANSPORTERS : INT;
END_VAR

VAR_EXTERNAL
  g_cfg : ARRAY[1..TRANSPORTERS] OF TRANSPORTER_CFG_T;
END_VAR
VAR
  ti   : INT;
  ai   : INT;
  area : TASK_AREA_T;
  can_lift : BOOL;
  can_sink : BOOL;
END_VAR

o_trans_id := 0;
FOR ti := 1 TO TRANSPORTERS DO
  IF o_trans_id = 0 THEN
    FOR ai := 1 TO 4 DO
      IF o_trans_id = 0 THEN
        area := g_cfg[ti].task_area[ai];
        IF area.min_lift > 0 OR area.max_lift > 0 THEN
          can_lift := (i_lift_stn >= area.min_lift) AND (i_lift_stn <= area.max_lift);
          IF i_sink_stn = 0 THEN
            (* Lift-only coverage search *)
            IF can_lift THEN
              o_trans_id := ti;
            END_IF;
          ELSE
            can_sink := (i_sink_stn >= area.min_sink) AND (i_sink_stn <= area.max_sink);
            IF can_lift AND can_sink THEN
              o_trans_id := ti;
            END_IF;
          END_IF;
        END_IF;
      END_IF;
    END_FOR;
  END_IF;
END_FOR;

END_FUNCTION_BLOCK

(* ---- STC_FB_MainScheduler.st ---- *)
(* ============================================================
   STC_FB_MainScheduler — Master scheduler orchestrator
   ============================================================
   Manages TSK_FB_Scheduler and DEP_FB_Scheduler calls on
   alternating PLC scan cycles. Ensures they never execute
   on the same cycle.

   Synchronization rules:
     1. Normal: alternate TSK_TURN → DEP_TURN → TSK_TURN ...
     2. Skip DEP when TSK is still computing (phase < 10000)
        → DEP would only sit in WAIT_STABLE anyway
     3. Skip DEP when g_dep_pending.valid = TRUE
        → TSK must process the pending data first
     4. g_dep_stable is computed internally after each TSK call

   Turn values:
     0 = INIT (first scan)
     1 = TSK_TURN  (TSK called this cycle)
     2 = DEP_TURN  (DEP called this cycle)

   Inputs:
     i_run     — enable (FALSE = both schedulers stopped)
     i_time_s  — absolute simulation time (seconds)

   Outputs:
     o_tsk_phase  — TSK current phase (forwarded)
     o_dep_phase  — DEP current phase (forwarded)
     o_turn       — which scheduler ran this cycle (1/2)
     o_skip_cnt   — DEP skip count (debug)
   ============================================================ *)

FUNCTION_BLOCK STC_FB_MainScheduler
VAR_INPUT
  i_run    : BOOL;     (* TRUE = run *)
  i_time_s : REAL;     (* current absolute time (s) *)
END_VAR
VAR_EXTERNAL
  g_dep_stable  : BOOL;
  g_dep_pending : DEP_PENDING_WRITE_T;
END_VAR
VAR_OUTPUT
  o_tsk_phase  : INT;     (* TSK scheduler phase *)
  o_dep_phase  : INT;     (* DEP scheduler phase *)
  o_turn       : INT;     (* 1=TSK ran, 2=DEP ran *)
  o_skip_cnt   : INT;     (* DEP skipped count (debug) *)
END_VAR
VAR
  tsk_sched    : TSK_FB_Scheduler;
  dep_sched    : DEP_FB_Scheduler;
  turn         : INT := 0;   (* 0=init, 1=TSK, 2=DEP *)
  skip_cnt     : INT := 0;
  tsk_phase    : INT := 0;
END_VAR

IF NOT i_run THEN
  (* Stop both schedulers *)
  tsk_sched(i_run := FALSE, i_time_s := 0.0);
  dep_sched(i_run := FALSE, i_time_s := 0.0, i_tsk_phase := 0);
  turn := 0;
  tsk_phase := 0;
  o_tsk_phase := 0;
  o_dep_phase := 0;
  o_turn := 0;
  RETURN;
END_IF;

(* ── Determine this cycle's turn ── *)
IF turn = 0 THEN
  (* First scan: always start with TSK *)
  turn := 1;

ELSIF turn = 1 THEN
  (* Last cycle was TSK → normally DEP's turn *)
  (* But skip DEP if: *)
  (*   a) TSK has not reached READY yet (phase < 10000) *)
  (*   b) pending data waiting for TSK to process *)
  IF tsk_phase < 10000 THEN
    (* TSK still computing — DEP would be blocked at WAIT_STABLE *)
    turn := 1;
    skip_cnt := skip_cnt + 1;
  ELSIF g_dep_pending.valid THEN
    (* TSK must process pending before DEP continues *)
    turn := 1;
    skip_cnt := skip_cnt + 1;
  ELSE
    turn := 2;
  END_IF;

ELSIF turn = 2 THEN
  (* Last cycle was DEP → TSK's turn *)
  turn := 1;
END_IF;

(* ── Execute the selected scheduler ── *)
IF turn = 1 THEN
  (* TSK turn *)
  tsk_sched(i_run := TRUE, i_time_s := i_time_s);
  tsk_phase := tsk_sched.o_phase;

  (* Compute stability flag after TSK call *)
  g_dep_stable := (tsk_phase >= 10000);

ELSIF turn = 2 THEN
  (* DEP turn *)
  dep_sched(
    i_run       := TRUE,
    i_time_s    := i_time_s,
    i_tsk_phase := tsk_phase
  );
END_IF;

(* ── Update outputs ── *)
o_tsk_phase := tsk_sched.o_phase;
o_dep_phase := dep_sched.o_phase;
o_turn      := turn;
o_skip_cnt  := skip_cnt;

END_FUNCTION_BLOCK

(* ---- STC_FB_MeasureMoveTimes.st ---- *)
(* ============================================================
   FB_TimeMoves → STC_FB_MeasureMoveTimes — Times actual transporter movements
   ============================================================
   Records real lift, sink, and travel times into g_move table
   by observing phase transitions in the transport cycle.
   Used by task scheduling and departure scheduling.

   Phase state machine (from plc_prg.st):
     0 → 1 : X-travel to lift station
     1 → 2 : Lift at station
     2 → 3 : X-travel to sink station
     3 → 4 : Sink at station
     4 → 0 : Cycle complete

   Filtering — only pure mechanical motion is timed:
     Travel (phase 1, 3): timer runs only when ABS(vel_x) > 0.1
       → filters out TWA collision avoidance stops.
     Lift (phase 2): timer runs only during z_stage 2, 3, 4
       → excludes device_delay + dropping_time (stage 1)
         and drip_delay (stage 5).
     Sink (phase 4): timer runs only during z_stage 7, 8
       → excludes device_delay + drip_delay (stage 6).

   Usage in plc_prg.st (one instance per transporter):
     tm1(t_id := 1, phase := g_transporter[1].phase,
         delta_t := 0.02, vel_x := g_transporter[1].vel_x,
         z_stage := g_transporter[1].z_stage,
         lift_stn := g_transporter[1].lift_station,
         sink_stn := g_transporter[1].sink_station,
         from_stn := g_transporter[1].current_station);

   Access recorded times:
     travel := g_move[1].travel[3].to_s[11];   stn 103 to 111
     lift   := g_move[1].lift_s[5];             lift at stn 105
     sink   := g_move[2].sink_s[12];            sink at stn 112
   ============================================================ *)

FUNCTION_BLOCK STC_FB_MeasureMoveTimes
VAR_INPUT
  t_id     : INT;     (* transporter index 1..3 *)
  phase    : INT;     (* current phase 0..4 *)
  delta_t  : REAL;    (* cycle time in seconds *)
  vel_x    : REAL;    (* current X velocity mm/s *)
  z_stage  : INT;     (* current Z motion stage 0..8 *)
  lift_stn : INT;     (* lift station number, e.g. 105 *)
  sink_stn : INT;     (* sink station number, e.g. 112 *)
  from_stn : INT;     (* station before command was given *)
END_VAR
VAR
  prev_phase   : INT := -1;   (* previous phase for edge detection *)
  timer        : REAL := 0.0; (* running timer *)
  travel_from  : INT;         (* index 1..25 for travel source *)
  travel_to    : INT;         (* index 1..25 for travel destination *)
  lift_idx     : INT;         (* index 1..25 for lift station *)
  sink_idx     : INT;         (* index 1..25 for sink station *)
END_VAR
VAR_EXTERNAL CONSTANT
    TRANSPORTERS : INT;
END_VAR

VAR_EXTERNAL
  g_move : ARRAY[1..TRANSPORTERS] OF MOVE_TIMES_T;
END_VAR

(* ---- Phase transition detection ---- *)
IF phase <> prev_phase THEN

  (* -- Save completed measurement and set up next -- *)

  IF prev_phase = 1 AND phase = 2 THEN
    (* Travel to lift complete → save travel time *)
    IF travel_from >= 1 AND travel_from <= 25
       AND travel_to >= 1 AND travel_to <= 25 THEN
      g_move[t_id].travel[travel_from].to_s[travel_to] := timer;
    END_IF;
    (* Start timing lift — timer starts at 0, accumulates only in z_stage 2-4 *)
    lift_idx := lift_stn - 100;
    timer := 0.0;

  ELSIF prev_phase = 2 AND phase = 3 THEN
    (* Lift complete → save lift time (pure mechanical Z-motion only) *)
    IF lift_idx >= 1 AND lift_idx <= 25 THEN
      g_move[t_id].lift_s[lift_idx] := timer;
    END_IF;
    (* Start timing travel to sink *)
    travel_from := lift_stn - 100;
    travel_to := sink_stn - 100;
    timer := 0.0;

  ELSIF prev_phase = 3 AND phase = 4 THEN
    (* Travel to sink complete → save travel time *)
    IF travel_from >= 1 AND travel_from <= 25
       AND travel_to >= 1 AND travel_to <= 25 THEN
      g_move[t_id].travel[travel_from].to_s[travel_to] := timer;
    END_IF;
    (* Start timing sink — timer starts at 0, accumulates only in z_stage 7-8 *)
    sink_idx := sink_stn - 100;
    timer := 0.0;

  ELSIF prev_phase = 4 AND phase = 0 THEN
    (* Sink complete → save sink time (pure mechanical Z-motion only) *)
    IF sink_idx >= 1 AND sink_idx <= 25 THEN
      g_move[t_id].sink_s[sink_idx] := timer;
    END_IF;
    timer := 0.0;

  ELSIF prev_phase = 0 AND phase = 1 THEN
    (* New cycle starting → set up travel-to-lift *)
    travel_from := from_stn - 100;
    travel_to := lift_stn - 100;
    timer := 0.0;

  ELSE
    (* Unexpected transition → just reset *)
    timer := 0.0;
  END_IF;

  prev_phase := phase;

ELSE
  (* ---- No transition: accumulate timer ---- *)

  IF phase = 1 OR phase = 3 THEN
    (* Travel: only count time when actually moving *)
    (* Filters out TWA collision avoidance stops    *)
    IF ABS(vel_x) > 0.1 THEN
      timer := timer + delta_t;
    END_IF;

  ELSIF phase = 2 THEN
    (* Lift: only mechanical Z-motion stages 2-4 *)
    (* Excludes: stage 1 (device_delay + dropping_time), stage 5 (drip_delay) *)
    IF z_stage >= 2 AND z_stage <= 4 THEN
      timer := timer + delta_t;
    END_IF;

  ELSIF phase = 4 THEN
    (* Sink: only mechanical Z-motion stages 7-8 *)
    (* Excludes: stage 6 (device_delay + drip_delay) *)
    IF z_stage >= 7 AND z_stage <= 8 THEN
      timer := timer + delta_t;
    END_IF;
  END_IF;

END_IF;

END_FUNCTION_BLOCK

(* ---- STC_FB_NoTreatmentStates.st ---- *)
(* ==========================================================
   STC_FB_NoTreatmentStates
   ----------------------------------------------------------
   Manages non-treatment target states for all units.

   Structure:
     Pass 0 — SNAPSHOT: read unit/batch/station state once into
              snap[] array. Also detects has_loading flag.
     Section 1 — PROCESSED: mark last-stage units as PROCESSED.
     Section 2 — TO_AVOID: clear occupied next-stage stations.
     Section 3 — TO_LOADING: route one empty unit to loading.
   ========================================================== *)

FUNCTION_BLOCK STC_FB_NoTreatmentStates
  VAR_EXTERNAL CONSTANT
    MAX_Units          : INT;
    MAX_STEPS_PER_PROGRAM         : INT;
    MAX_STATIONS_PER_STEP      : INT;
    MIN_StationIndex : INT;
    MAX_StationIndex  : INT;
    IN_PROCESS         : INT;
    PROCESSED          : INT;
    NOT_USED           : INT;
    TO_NONE            : INT;
    TO_AVOID           : INT;
    TO_LOADING         : INT;
    USED               : INT;
    OP_LOADING           : INT;
    OP_LOADING_UNLOADING : INT;
  END_VAR

  VAR_EXTERNAL
    g_unit             : ARRAY[1..MAX_Units] OF UNIT_T;
    g_batch            : ARRAY[1..MAX_Units] OF BATCH_T;
    g_program          : ARRAY[1..MAX_Units] OF TREATMENT_PROGRAM_T;
    g_station          : ARRAY[MIN_StationIndex..MAX_StationIndex] OF UDT_StationType;
    g_time_s           : LINT;
    g_production_queue : INT;
  END_VAR

  VAR
    (* Snapshot *)
    snap        : ARRAY[1..MAX_Units] OF UNIT_SNAP_T;
    u           : INT;        (* unit loop index *)
    has_loading : BOOL;       (* any unit already has TO_LOADING *)
    (* Section 1+2 *)
    p           : INT;        (* parallel station loop *)
    next_stn    : INT;        (* next stage station *)
    occ_uid     : INT;        (* unit_id at an occupied station *)
    free_found  : BOOL;       (* any next-stage station is free *)
    avoid_uid   : INT;        (* unit to mark TO_AVOID *)
    (* Section 3 *)
    load_free   : BOOL;       (* a loading station is free *)
    load_uid    : INT;        (* best candidate for TO_LOADING *)
    load_in_buf : BOOL;       (* current candidate is in buffer *)
    stk         : INT;        (* station loop *)
    op          : INT;        (* station operation code *)
  END_VAR

  (* ════════════════════════════════════════════════════════════
     Pass 0 — SNAPSHOT: collect per-unit state in one pass
     ════════════════════════════════════════════════════════════ *)
  has_loading := FALSE;

  FOR u := 1 TO MAX_Units DO
    snap[u].active := g_unit[u].status <> NOT_USED;
    IF NOT snap[u].active THEN
      CONTINUE;
    END_IF;

    snap[u].loc       := g_unit[u].location;
    snap[u].tgt       := g_unit[u].target;
    snap[u].has_batch := g_batch[u].batch_code <> 0;
    snap[u].bstate    := g_batch[u].state;
    snap[u].cur_stage := g_batch[u].cur_stage;

    snap[u].on_station := snap[u].loc >= MIN_StationIndex
                          AND snap[u].loc <= MAX_StationIndex;
    IF snap[u].on_station THEN
      snap[u].loc_op    := g_station[snap[u].loc].StationType;
      snap[u].in_buffer := snap[u].loc_op >= 44 AND snap[u].loc_op <= 47;
      IF g_station[snap[u].loc].ChangeTime > 0 THEN
        snap[u].elapsed := g_time_s - g_station[snap[u].loc].ChangeTime;
      ELSE
        snap[u].elapsed := 0;
      END_IF;
      snap[u].cal := g_program[u].stages[snap[u].cur_stage].cal_time;
    ELSE
      snap[u].loc_op    := 0;
      snap[u].in_buffer := FALSE;
      snap[u].elapsed   := 0;
      snap[u].cal       := 0;
    END_IF;

    IF snap[u].tgt = TO_LOADING THEN
      has_loading := TRUE;
    END_IF;
  END_FOR;

  (* ════════════════════════════════════════════════════════════
     Section 1 — PROCESSED: mark batch done at last treatment stage
     ════════════════════════════════════════════════════════════
     For each IN_PROCESS unit on a station:
       If next stage is empty (stations[1]=0) → last stage.
       If elapsed >= cal_time → set state := PROCESSED. *)
  FOR u := 1 TO MAX_Units DO
    IF NOT snap[u].active OR NOT snap[u].has_batch THEN
      CONTINUE;
    END_IF;
    IF snap[u].bstate <> IN_PROCESS OR NOT snap[u].on_station THEN
      CONTINUE;
    END_IF;
    IF snap[u].cur_stage >= 1 AND snap[u].cur_stage < MAX_STEPS_PER_PROGRAM THEN
      IF g_program[u].stages[snap[u].cur_stage + 1].stations[1] = 0 THEN
        IF snap[u].elapsed > 0 AND snap[u].elapsed >= DINT_TO_LINT(snap[u].cal) THEN
          g_batch[u].state := PROCESSED;
          snap[u].bstate   := PROCESSED;  (* update snapshot *)
        END_IF;
      END_IF;
    END_IF;
  END_FOR;

  (* ════════════════════════════════════════════════════════════
     Section 2 — TO_AVOID: clear the way to next treatment station
     ════════════════════════════════════════════════════════════
     For each IN_PROCESS unit whose next stage exists:
       Pass 1: check if any next-stage station is free or already
               has a TO_AVOID unit (slot being cleared).
       Pass 2: if all occupied, mark ONE empty-batch TO_NONE unit
               at those stations as TO_AVOID. *)
  FOR u := 1 TO MAX_Units DO
    IF NOT snap[u].active OR NOT snap[u].has_batch THEN
      CONTINUE;
    END_IF;
    IF snap[u].bstate <> IN_PROCESS THEN
      CONTINUE;
    END_IF;
    IF snap[u].cur_stage < 1 OR snap[u].cur_stage >= MAX_STEPS_PER_PROGRAM THEN
      CONTINUE;
    END_IF;
    IF g_program[u].stages[snap[u].cur_stage + 1].stations[1] = 0 THEN
      CONTINUE;  (* no next stage *)
    END_IF;

    (* — Pass 1: any next-stage station free or being cleared? — *)
    free_found := FALSE;
    avoid_uid  := 0;
    FOR p := 1 TO MAX_STATIONS_PER_STEP DO
      next_stn := g_program[u].stages[snap[u].cur_stage + 1].stations[p];
      IF next_stn = 0 THEN
        EXIT;
      END_IF;
      IF next_stn >= MIN_StationIndex AND next_stn <= MAX_StationIndex THEN
        IF g_station[next_stn].UnitId = 0 THEN
          free_found := TRUE;
          EXIT;
        END_IF;
        occ_uid := g_station[next_stn].UnitId;
        IF occ_uid >= 1 AND occ_uid <= MAX_Units THEN
          IF snap[occ_uid].tgt = TO_AVOID THEN
            free_found := TRUE;
            EXIT;
          END_IF;
        END_IF;
      END_IF;
    END_FOR;

    (* — Pass 2: all occupied → mark ONE movable unit TO_AVOID — *)
    IF NOT free_found THEN
      FOR p := 1 TO MAX_STATIONS_PER_STEP DO
        next_stn := g_program[u].stages[snap[u].cur_stage + 1].stations[p];
        IF next_stn = 0 THEN
          EXIT;
        END_IF;
        IF next_stn >= MIN_StationIndex AND next_stn <= MAX_StationIndex THEN
          occ_uid := g_station[next_stn].UnitId;
          IF occ_uid >= 1 AND occ_uid <= MAX_Units THEN
            IF NOT snap[occ_uid].has_batch AND snap[occ_uid].tgt = TO_NONE THEN
              avoid_uid := occ_uid;
              EXIT;
            END_IF;
          END_IF;
        END_IF;
      END_FOR;

      IF avoid_uid >= 1 THEN
        g_unit[avoid_uid].target := TO_AVOID;
        snap[avoid_uid].tgt     := TO_AVOID;  (* update snapshot *)
      END_IF;
    END_IF;
  END_FOR;

  (* ════════════════════════════════════════════════════════════
     Section 3 — TO_LOADING: route one empty unit to loading station
     ════════════════════════════════════════════════════════════
     When production is active and a loading/loading_unloading station
     is free, find ONE batchless USED unit with TO_NONE target.
     Priority: units NOT in buffer/storage first. *)
  IF g_production_queue = 1 AND NOT has_loading THEN

    (* Check if any loading station is free *)
    load_free := FALSE;
    FOR stk := MIN_StationIndex TO MAX_StationIndex DO
      op := g_station[stk].StationType;
      IF (op = OP_LOADING OR op = OP_LOADING_UNLOADING)
         AND g_station[stk].UnitId = 0 THEN
        load_free := TRUE;
        EXIT;
      END_IF;
    END_FOR;

    IF load_free THEN
      load_uid    := 0;
      load_in_buf := FALSE;
      FOR u := 1 TO MAX_Units DO
        IF snap[u].active AND NOT snap[u].has_batch
           AND snap[u].tgt = TO_NONE AND snap[u].on_station THEN
          IF snap[u].in_buffer THEN
            IF load_uid = 0 THEN
              load_uid    := u;
              load_in_buf := TRUE;
            END_IF;
          ELSE
            IF load_uid = 0 OR load_in_buf THEN
              load_uid    := u;
              load_in_buf := FALSE;
            END_IF;
          END_IF;
        END_IF;
      END_FOR;

      IF load_uid >= 1 THEN
        g_unit[load_uid].target := TO_LOADING;
      END_IF;
    END_IF; (* load_free *)

  END_IF; (* production_queue AND NOT has_loading *)

END_FUNCTION_BLOCK

(* ---- STC_FB_ShiftSchedule.st ---- *)
(* ============================================================
   STC_FB_ShiftSchedule — Shift schedule + task times
   ============================================================
   Propagates a time shift through one unit's schedule stages
   AND through all matching tasks in the 3 transporter queues.

   Positive i_amount = DELAY (shift later),
   Negative i_amount = ADVANCE (shift earlier).

   Replaces 4× duplicated propagation code in TSK_FB_Resolve.
   ============================================================ *)

FUNCTION_BLOCK STC_FB_ShiftSchedule
VAR_INPUT
  i_unit       : INT;     (* unit index 1..10 *)
  i_from_stage : INT;     (* propagate from this stage onward *)
  i_amount     : REAL;    (* seconds to shift (+ = later, - = earlier) *)
END_VAR
VAR_EXTERNAL CONSTANT
    TRANSPORTERS : INT;
END_VAR

VAR_EXTERNAL
  g_schedule : ARRAY[1..10] OF TSK_SCHEDULE_T;
  g_tasks    : ARRAY[1..TRANSPORTERS] OF TSK_QUEUE_T;
END_VAR
VAR
  sc : INT;
  si : INT;
  qi : INT;
  ti : INT;
END_VAR

IF i_unit < 1 OR i_unit > 10 THEN RETURN; END_IF;
IF ABS(i_amount) < 0.001 THEN RETURN; END_IF;

(* ── Shift schedule stages entry/exit times ── *)
sc := g_schedule[i_unit].stage_count;
FOR si := i_from_stage TO sc DO
  IF si >= 1 AND si <= 30 THEN
    g_schedule[i_unit].stages[si].entry_time :=
      g_schedule[i_unit].stages[si].entry_time + REAL_TO_LINT(i_amount);
    g_schedule[i_unit].stages[si].exit_time :=
      g_schedule[i_unit].stages[si].exit_time + REAL_TO_LINT(i_amount);
  END_IF;
END_FOR;

(* ── Shift matching tasks in all transporter queues ── *)
FOR ti := 1 TO TRANSPORTERS DO
  FOR qi := 1 TO g_tasks[ti].count DO
    IF g_tasks[ti].queue[qi].unit = i_unit
       AND g_tasks[ti].queue[qi].stage >= i_from_stage THEN
      g_tasks[ti].queue[qi].start_time :=
        g_tasks[ti].queue[qi].start_time + REAL_TO_LINT(i_amount);
      g_tasks[ti].queue[qi].finish_time :=
        g_tasks[ti].queue[qi].finish_time + REAL_TO_LINT(i_amount);
    END_IF;
  END_FOR;
END_FOR;

END_FUNCTION_BLOCK

(* ---- STC_FB_SortTaskQueue.st ---- *)
(* ============================================================
   STC_FB_SortTaskQueue — Insertion sort task queues by start_time
   ============================================================
   Sorts one or all transporter task queues in-place using
   insertion sort (stable, O(n²) — fine for n ≤ 10).

   Mode controlled by i_trans:
     0   = sort ALL queues (1..3)
     1-3 = sort only that transporter's queue

   Replaces 3× duplicated insertion sort code in:
     TSK_FB_Scheduler (phase 2200)
     DEP_FB_Scheduler (phase 1020)
     TSK_FB_Analyze   (merge-sort variant — still inline)
   ============================================================ *)

FUNCTION_BLOCK STC_FB_SortTaskQueue
VAR_INPUT
  i_trans : INT;    (* 0 = all, 1..3 = specific transporter *)
END_VAR
VAR_EXTERNAL CONSTANT
    TRANSPORTERS : INT;
END_VAR

VAR_EXTERNAL
  g_tasks : ARRAY[1..TRANSPORTERS] OF TSK_QUEUE_T;
END_VAR
VAR
  ti       : INT;
  t_start  : INT;
  t_end    : INT;
  ins_i    : INT;
  ins_j    : INT;
  ins_cnt  : INT;
  tmp_task : TSK_TASK_T;
END_VAR

IF i_trans >= 1 AND i_trans <= 3 THEN
  t_start := i_trans;
  t_end   := i_trans;
ELSE
  t_start := 1;
  t_end   := 3;
END_IF;

FOR ti := t_start TO t_end DO
  ins_cnt := g_tasks[ti].count;
  IF ins_cnt >= 2 THEN
    FOR ins_i := 2 TO ins_cnt DO
      tmp_task := g_tasks[ti].queue[ins_i];
      ins_j := ins_i - 1;
      WHILE ins_j >= 1 AND g_tasks[ti].queue[ins_j].start_time > tmp_task.start_time DO
        g_tasks[ti].queue[ins_j + 1] := g_tasks[ti].queue[ins_j];
        ins_j := ins_j - 1;
      END_WHILE;
      g_tasks[ti].queue[ins_j + 1] := tmp_task;
    END_FOR;
  END_IF;
END_FOR;

END_FUNCTION_BLOCK

(* ---- STC_FB_UpdateUnitLocation.st ---- *)
(* ============================================================
   STC_FB_UpdateUnitLocation — Update a unit's location
   ============================================================
   Sets g_unit[i_unit].location to the given new location.
   Location < 100 = transporter, >= 100 = station.
   Updates unit_id + change_time on the relevant station(s).

   When moving to a station (sink / task completion):
     - Advances batch cur_stage if batch is IN_PROCESS
     - Updates batch min_time/max_time/cal_time from treatment program
     - Clears unit target to TO_NONE if target was set (NTT done)
   ============================================================ *)

FUNCTION_BLOCK STC_FB_UpdateUnitLocation
VAR_INPUT
  i_unit     : INT;   (* unit number to update *)
  i_location : INT;   (* new location: <100 = transporter id, >=100 = station number *)
END_VAR
VAR_EXTERNAL CONSTANT
    MAX_UNITS           : INT;
    MAX_TRANSPORTERS    : INT;
    MAX_STAGES          : INT;
    STATION_ARRAY_START : INT;
    STATION_ARRAY_END   : INT;
    IN_PROCESS          : INT;
END_VAR
VAR_EXTERNAL
  g_unit        : ARRAY[1..MAX_UNITS] OF UNIT_T;
  g_station     : ARRAY[STATION_ARRAY_START..STATION_ARRAY_END] OF STATION_T;
  g_transporter : ARRAY[1..MAX_TRANSPORTERS] OF STC_TRANSPORTER_T;
  g_batch       : ARRAY[1..MAX_UNITS] OF BATCH_T;
  g_program     : ARRAY[1..MAX_UNITS] OF TREATMENT_PROGRAM_T;
  g_time_s      : LINT;
END_VAR
VAR
  old_loc : INT;
  new_stg : INT;
END_VAR

IF (i_unit >= 1) AND (i_unit <= MAX_UNITS) THEN
  old_loc := g_unit[i_unit].location;

  (* --- Clear unit_id from old location --- *)
  IF (old_loc >= STATION_ARRAY_START) AND (old_loc <= STATION_ARRAY_END) THEN
    (* Was on a station — clear station unit_id, stamp change_time *)
    g_station[old_loc].unit_id     := 0;
    g_station[old_loc].change_time := g_time_s;
  ELSIF (old_loc >= 1) AND (old_loc <= MAX_TRANSPORTERS) THEN
    (* Was on a transporter — clear transporter unit_id *)
    g_transporter[old_loc].unit_id := 0;
  END_IF;

  (* --- Update unit location --- *)
  g_unit[i_unit].location := i_location;

  (* --- Set unit_id on new location --- *)
  IF (i_location >= STATION_ARRAY_START) AND (i_location <= STATION_ARRAY_END) THEN
    (* Moving to a station (sink completion) *)
    g_station[i_location].unit_id     := i_unit;
    g_station[i_location].change_time := g_time_s;

    (* Advance batch stage if unit is USED with an active batch *)
    IF (g_unit[i_unit].status = 1)  (* USED *)
       AND (g_batch[i_unit].batch_code <> 0)
       AND (g_batch[i_unit].state = IN_PROCESS)
       AND (g_batch[i_unit].cur_stage < MAX_STAGES) THEN
      g_batch[i_unit].cur_stage := g_batch[i_unit].cur_stage + 1;

      (* Stamp arrival time on new station — used by CalcSchedule for elapsed calculation *)
      g_batch[i_unit].start_time := g_time_s;

      (* Update batch treatment times from program for the new stage *)
      IF (g_program[i_unit].program_id = g_batch[i_unit].prog_id)
         AND (g_program[i_unit].program_id > 0) THEN
        new_stg := g_batch[i_unit].cur_stage;
        IF (new_stg >= 1) AND (new_stg <= MAX_STAGES) THEN
          g_batch[i_unit].min_time := g_program[i_unit].stages[new_stg].min_time;
          g_batch[i_unit].max_time := g_program[i_unit].stages[new_stg].max_time;
          g_batch[i_unit].cal_time := g_program[i_unit].stages[new_stg].cal_time;
        END_IF;
      END_IF;
    END_IF;

    (* NOT_PROCESSED batch on station: clear times so UI shows no progress bar *)
    IF (g_batch[i_unit].batch_code <> 0)
       AND (g_batch[i_unit].state <> IN_PROCESS) THEN
      g_batch[i_unit].min_time   := 0;
      g_batch[i_unit].cal_time   := 0;
      g_batch[i_unit].max_time   := 32000;  (* ~8.9 h cap, INT max safe *)
      g_batch[i_unit].start_time := g_time_s;
    END_IF;

    (* Clear unit target after placement (NTT task done) *)
    IF g_unit[i_unit].target <> 0 THEN
      g_unit[i_unit].target := 0;  (* TO_NONE *)
    END_IF;

  ELSIF (i_location >= 1) AND (i_location <= MAX_TRANSPORTERS) THEN
    (* Moving to a transporter (lift start) *)
    g_transporter[i_location].unit_id := i_unit;
  END_IF;
END_IF;

END_FUNCTION_BLOCK

(* ---- STC_FindTransporter.st ---- *)
(* ============================================================
   STC_FindTransporter — Find covering transporter (FB)
   ============================================================
   Finds which transporter (1..3) can handle a lift→sink pair
   by checking cfg[].TaskArea[] coverage.

   If i_sink_stn = 0, only lift coverage is checked (used when
   looking for the transporter covering a single station).

   NOTE: Kept as FUNCTION_BLOCK because MATIEC's C code generator
   cannot handle ARRAY OF STRUCT as FUNCTION VAR_INPUT parameter.
   (C++ __SET_VAR macro produces type mismatch.)

   Used by: TSK_FB_CreateTasks, TSK_FB_Scheduler, DEP_FB_Scheduler
   ============================================================ *)

FUNCTION_BLOCK STC_FindTransporter
VAR_INPUT
  i_lift_stn : INT;     (* lift station number *)
  i_sink_stn : INT;     (* sink station number, 0 = lift-only search *)
END_VAR
VAR_OUTPUT
  o_trans : INT;         (* transporter ID 1..3, 0 = not found *)
END_VAR
VAR_EXTERNAL CONSTANT
  MAX_Transporters : INT;
END_VAR
VAR_EXTERNAL
  g_cfg : ARRAY[1..MAX_Transporters] OF UDT_TransporterType;
END_VAR
VAR
  ti       : INT;
  ai       : INT;
  area     : UDT_TaskArea;
  can_lift : BOOL;
  can_sink : BOOL;
END_VAR

o_trans := 0;
FOR ti := 1 TO MAX_Transporters DO
  IF o_trans = 0 THEN
    FOR ai := 1 TO 4 DO
      IF o_trans = 0 THEN
        area := g_cfg[ti].TaskArea[ai];
        IF area.MinLift > 0 OR area.MaxLift > 0 THEN
          can_lift := (i_lift_stn >= area.MinLift) AND (i_lift_stn <= area.MaxLift);
          IF i_sink_stn = 0 THEN
            IF can_lift THEN
              o_trans := ti;
            END_IF;
          ELSE
            can_sink := (i_sink_stn >= area.MinSink) AND (i_sink_stn <= area.MaxSink);
            IF can_lift AND can_sink THEN
              o_trans := ti;
            END_IF;
          END_IF;
        END_IF;
      END_IF;
    END_FOR;
  END_IF;
END_FOR;

END_FUNCTION_BLOCK
